  MoveL 7109 to (-196.28, 113.55, -59.38) mm, rotated rx -180 ry 0 rz 0.01 deg; joints [33.121, -44.409, 105.937, -143.593, 67.066, 164.943]
  MoveL 7110 to (-202.77, 114.78, -59.62) mm, rotated rx 180 ry 0 rz 0.01 deg; joints [33.024, -44.143, 105.375, -143.62, 66.8, 164.793]
  MoveL 7111 to (-206.5, 109.33, -59.86) mm, rotated rx 180 ry 0 rz 0.01 deg; joints [32.769, -44.118, 105.358, -143.888, 66.734, 164.906]
  MoveL 7112 to (-202.99, 103.73, -60.11) mm, rotated rx -180 ry 0 rz 0.01 deg; joints [32.66, -44.348, 105.903, -144.081, 66.958, 165.153]
  MoveL 7113 to (-196.46, 104.7, -60.35) mm, rotated rx 180 ry 0 rz 0.01 deg; joints [32.829, -44.542, 106.356, -143.969, 67.215, 165.248]
  MoveL 7114 to (-194.73, 111.07, -60.6) mm, rotated rx 180 ry 0 rz 0.01 deg; joints [33.074, -44.451, 106.172, -143.69, 67.208, 165.087]
  MoveL 7115 to (-199.87, 115.21, -60.84) mm, rotated rx 180 ry 0 rz 0.01 deg; joints [33.1, -44.169, 105.569, -143.583, 66.956, 164.869]
  MoveL 7116 to (-205.73, 112.16, -61.08) mm, rotated rx 180 ry 0 rz 0.01 deg; joints [32.878, -44.018, 105.268, -143.777, 66.773, 164.866]
  MoveL 7117 to (-205.28, 105.57, -61.33) mm, rotated rx -180 ry 0 rz 0.01 deg; joints [32.673, -44.163, 105.628, -144.045, 66.889, 165.09]
  MoveL 7118 to (-199.06, 103.34, -61.57) mm, rotated rx 180 ry 0 rz 0.01 deg; joints [32.731, -44.414, 106.215, -144.068, 67.177, 165.28]
  MoveL 7119 to (-194.53, 108.15, -61.82) mm, rotated rx 180 ry 0 rz 0.01 deg; joints [32.984, -44.455, 106.324, -143.821, 67.302, 165.219]
  MoveL 7120 to (-197.11, 114.22, -62.06) mm, rotated rx 180 ry 0 rz 0.01 deg; joints [33.127, -44.221, 105.822, -143.606, 67.126, 164.988]
  MoveL 7121 to (-203.72, 114.29, -62.3) mm, rotated rx 180 ry 0 rz 0.01 deg; joints [32.99, -43.977, 105.309, -143.681, 66.871, 164.872]
  MoveL 7122 to (-206.42, 108.27, -62.55) mm, rotated rx -180 ry 0 rz 0.01 deg; joints [32.737, -43.999, 105.398, -143.961, 66.853, 165.021]
  MoveL 7123 to (-201.99, 103.37, -62.79) mm, rotated rx -180 ry 0 rz 0.01 deg; joints [32.671, -44.246, 105.98, -144.114, 67.106, 165.263]
  MoveL 7124 to (-195.73, 105.47, -63.04) mm, rotated rx 180 ry 0 rz 0.01 deg; joints [32.871, -44.405, 106.356, -143.958, 67.337, 165.318]
  MoveL 7125 to (-195.14, 112.05, -63.28) mm, rotated rx 180 ry 0 rz 0.01 deg; joints [33.099, -44.27, 106.072, -143.685, 67.28, 165.129]
  MoveL 7126 to (-200.94, 115.22, -63.52) mm, rotated rx 180 ry 0 rz 0.01 deg; joints [33.079, -43.988, 105.468, -143.625, 67.016, 164.93]
  MoveL 7127 to (-206.16, 111.18, -63.77) mm, rotated rx -180 ry 0 rz 0.01 deg; joints [32.838, -43.88, 105.264, -143.852, 66.87, 164.969]
  MoveL 7128 to (-204.56, 104.78, -64.01) mm, rotated rx 180 ry 0 rz 0.01 deg; joints [32.664, -44.06, 105.704, -144.099, 67.031, 165.208]
  MoveL 7129 to (-198.05, 103.68, -64.26) mm, rotated rx 180 ry 0 rz 0.01 deg; joints [32.765, -44.297, 106.258, -144.072, 67.316, 165.368]
  MoveL 7130 to (-194.43, 109.21, -64.5) mm, rotated rx 180 ry 0 rz 0.01 deg; joints [33.022, -44.29, 106.26, -143.807, 67.394, 165.268]
  MoveC 7131 to (-196.76, 111.53, -64.5) mm, rotated rx 180 ry 0 rz 0.01 deg; joints [33.048, -44.16, 105.966, -143.739, 67.27, 165.152] to (-199.08, 109.21, -64.5) mm, rotated rx 180 ry 0 rz 0.01 deg; joints [32.923, -44.129, 105.903, -143.861, 67.209, 165.183]
  MoveC 7132 to (-196.76, 106.88, -64.5) mm, rotated rx 180 ry 0 rz 0.01 deg; joints [32.897, -44.26, 106.197, -143.929, 67.333, 165.299] to (-194.43, 109.21, -64.5) mm, rotated rx -180 ry 0 rz 0.01 deg; joints [33.022, -44.29, 106.26, -143.807, 67.394, 165.268]
  MoveC 7133 to (-193.87, 111.26, -64.5) mm, rotated rx 180 ry 0 rz 0.01 deg; joints [33.1, -44.265, 106.201, -143.716, 67.389, 165.214] to (-192.35, 112.73, -64.5) mm, rotated rx -180 ry 0 rz 0.01 deg; joints [33.181, -44.286, 106.244, -143.638, 67.429, 165.195]
  MoveC 7134 to (-191.13, 114.78, -64.5) mm, rotated rx -180 ry 0 rz 0.01 deg; joints [33.273, -44.283, 106.235, -143.54, 67.449, 165.153] to (-192.33, 116.83, -64.5) mm, rotated rx -180 ry 0 rz 0.01 deg; joints [33.315, -44.198, 106.04, -143.471, 67.374, 165.066]
  MoveC 7135 to (-193.08, 117.28, -64.5) mm, rotated rx -180 ry 0 rz 0.01 deg; joints [33.313, -44.162, 105.96, -143.461, 67.337, 165.038] to (-193.81, 117.76, -64.5) mm, rotated rx -180 ry 0 rz 0.01 deg; joints [33.313, -44.126, 105.88, -143.45, 67.302, 165.009]
  MoveC 7136 to (-196.76, 118.7, -64.5) mm, rotated rx -180 ry 0 rz 0.01 deg; joints [33.281, -44.004, 105.608, -143.446, 67.172, 164.926] to (-199.7, 117.76, -64.5) mm, rotated rx 180 ry 0 rz 0.01 deg; joints [33.188, -43.923, 105.429, -143.518, 67.067, 164.901]
  MoveC 7137 to (-201.1, 116.87, -64.5) mm, rotated rx 180 ry 0 rz 0.01 deg; joints [33.13, -43.893, 105.365, -143.57, 67.023, 164.904] to (-202.59, 116.12, -64.5) mm, rotated rx 180 ry 0 rz 0.01 deg; joints [33.074, -43.858, 105.289, -143.618, 66.974, 164.9]
  MoveC 7138 to (-204.95, 114.01, -64.5) mm, rotated rx -180 ry 0 rz 0.01 deg; joints [32.956, -43.821, 105.212, -143.731, 66.908, 164.924] to (-205.64, 110.92, -64.5) mm, rotated rx 180 ry 0 rz 0.01 deg; joints [32.841, -43.864, 105.313, -143.865, 66.923, 165.009]
  MoveC 7139 to (-205.56, 109.27, -64.5) mm, rotated rx -180 ry 0 rz 0.01 deg; joints [32.789, -43.903, 105.401, -143.932, 66.948, 165.063] to (-205.65, 107.61, -64.5) mm, rotated rx -180 ry 0 rz 0.01 deg; joints [32.733, -43.935, 105.476, -144.001, 66.967, 165.113]
  MoveC 7140 to (-205, 104.51, -64.5) mm, rotated rx 180 ry 0 rz 0.01 deg; joints [32.646, -44.024, 105.68, -144.12, 67.036, 165.223] to (-202.66, 102.37, -64.5) mm, rotated rx -180 ry 0 rz 0.01 deg; joints [32.625, -44.151, 105.966, -144.182, 67.158, 165.333]
  MoveC 7141 to (-201.23, 101.62, -64.5) mm, rotated rx -180 ry 0 rz 0.01 deg; joints [32.63, -44.217, 106.113, -144.196, 67.226, 165.382] to (-199.87, 100.74, -64.5) mm, rotated rx 180 ry 0 rz 0.01 deg; joints [32.63, -44.283, 106.261, -144.217, 67.293, 165.434]
  MoveC 7142 to (-196.86, 99.74, -64.5) mm, rotated rx 180 ry 0 rz 0.01 deg; joints [32.66, -44.408, 106.541, -144.223, 67.427, 165.52] to (-193.81, 100.62, -64.5) mm, rotated rx -180 ry 0 rz 0.01 deg; joints [32.754, -44.494, 106.731, -144.151, 67.536, 165.547]
  MoveC 7143 to (-193.08, 101.1, -64.5) mm, rotated rx -180 ry 0 rz 0.01 deg; joints [32.785, -44.509, 106.763, -144.122, 67.559, 165.546] to (-192.33, 101.56, -64.5) mm, rotated rx 180 ry 0 rz 0.01 deg; joints [32.816, -44.525, 106.798, -144.095, 67.582, 165.545]
  MoveC 7144 to (-191.57, 102, -64.5) mm, rotated rx 180 ry 0 rz 0.01 deg; joints [32.846, -44.542, 106.834, -144.068, 67.607, 165.545] to (-190.79, 102.39, -64.5) mm, rotated rx 180 ry 0 rz 0.01 deg; joints [32.876, -44.561, 106.875, -144.042, 67.632, 165.547]
  MoveC 7145 to (-188.5, 104.54, -64.5) mm, rotated rx -180 ry 0 rz 0.01 deg; joints [32.995, -44.594, 106.944, -143.927, 67.694, 165.521] to (-187.86, 107.61, -64.5) mm, rotated rx -180 ry 0 rz 0.01 deg; joints [33.109, -44.55, 106.841, -143.794, 67.677, 165.437]
  MoveC 7146 to (-187.95, 109.27, -64.5) mm, rotated rx -180 ry 0 rz 0.01 deg; joints [33.162, -44.511, 106.752, -143.727, 67.651, 165.384] to (-187.87, 110.92, -64.5) mm, rotated rx -180 ry 0 rz 0.01 deg; joints [33.217, -44.478, 106.675, -143.659, 67.631, 165.333]
  MoveC 7147 to (-188.56, 114.01, -64.5) mm, rotated rx 180 ry 0 rz 0.01 deg; joints [33.304, -44.388, 106.469, -143.541, 67.562, 165.224] to (-190.92, 116.12, -64.5) mm, rotated rx 180 ry 0 rz 0.01 deg; joints [33.322, -44.261, 106.183, -143.483, 67.439, 165.114]
  MoveC 7148 to (-191.64, 116.46, -64.5) mm, rotated rx -180 ry 0 rz 0.01 deg; joints [33.318, -44.23, 106.112, -143.477, 67.406, 165.09] to (-192.33, 116.83, -64.5) mm, rotated rx 180 ry 0 rz 0.01 deg; joints [33.315, -44.198, 106.04, -143.471, 67.374, 165.066]
  MoveL 7149 to (-192.94, 116.99, -64.33) mm, rotated rx -180 ry 0 rz 0.01 deg; joints [33.307, -44.183, 105.987, -143.469, 67.341, 165.045]
  MoveL 7150 to (-193.39, 116.91, -63.87) mm, rotated rx 180 ry 0 rz 0.01 deg; joints [33.294, -44.194, 105.96, -143.473, 67.306, 165.025]
  MoveL 7151 to (-193.55, 116.84, -63.23) mm, rotated rx -180 ry 0 rz 0.01 deg; joints [33.288, -44.224, 105.956, -143.47, 67.277, 165.005]
  Set speed (1000.0 mm/s)
  MoveL 7152 to (-193.55, 116.84, 11) mm, rotated rx 180 ry 0 rz 0.01 deg; joints [33.247, -48.144, 106.249, -142.533, 64.368, 162.631]
  Set speed (1000.0 mm/s)
  MoveL 7153 to (-195.99, 9.51, 11) mm, rotated rx 180 ry 0 rz 0.01 deg; joints [29.569, -50.402, 111.087, -147.115, 65.397, 165.962]
  Set speed (1000.0 mm/s)
  MoveL 7154 to (-195.99, 9.51, -42.73) mm, rotated rx -180 ry 0 rz 0.01 deg; joints [29.603, -47.446, 110.916, -147.729, 67.753, 167.582]
  Set speed (100.0 mm/s)
  MoveL 7155 to (-196.15, 9.53, -43.35) mm, rotated rx 180 ry 0 rz 0.01 deg; joints [29.601, -47.405, 110.899, -147.736, 67.773, 167.597]
  MoveL 7156 to (-196.59, 9.56, -43.82) mm, rotated rx 180 ry 0 rz 0.01 deg; joints [29.593, -47.363, 110.861, -147.745, 67.774, 167.603]
  MoveL 7157 to (-197.21, 9.55, -44) mm, rotated rx 180 ry 0 rz 0.01 deg; joints [29.58, -47.331, 110.814, -147.755, 67.758, 167.598]
  MoveL 7158 to (-202.45, 5.52, -44.24) mm, rotated rx 180 ry 0 rz 0.01 deg; joints [29.336, -47.21, 110.584, -147.988, 67.608, 167.636]
  MoveL 7159 to (-200.86, -0.89, -44.49) mm, rotated rx 180 ry 0 rz 0.01 deg; joints [29.142, -47.371, 110.981, -148.243, 67.762, 167.85]
  MoveL 7160 to (-194.35, -2, -44.73) mm, rotated rx 180 ry 0 rz 0.01 deg; joints [29.231, -47.605, 111.527, -148.216, 68.049, 167.992]
  MoveL 7161 to (-190.72, 3.52, -44.98) mm, rotated rx -180 ry 0 rz 0.01 deg; joints [29.498, -47.615, 111.567, -147.942, 68.136, 167.901]
  MoveL 7162 to (-194.32, 9.05, -45.22) mm, rotated rx 180 ry 0 rz 0.01 deg; joints [29.621, -47.373, 111.05, -147.754, 67.932, 167.694]
  MoveL 7163 to (-200.84, 7.97, -45.46) mm, rotated rx 180 ry 0 rz 0.01 deg; joints [29.454, -47.152, 110.595, -147.879, 67.694, 167.627]
  MoveL 7164 to (-202.46, 1.57, -45.71) mm, rotated rx 180 ry 0 rz 0.01 deg; joints [29.198, -47.201, 110.746, -148.17, 67.72, 167.79]
  MoveL 7165 to (-197.24, -2.48, -45.95) mm, rotated rx -180 ry 0 rz 0.01 deg; joints [29.158, -47.444, 111.319, -148.283, 67.991, 167.994]
  MoveL 7166 to (-191.44, 0.67, -46.2) mm, rotated rx 180 ry 0 rz 0.01 deg; joints [29.384, -47.574, 111.627, -148.083, 68.195, 168.005]
  MoveL 7167 to (-192.01, 7.25, -46.44) mm, rotated rx -180 ry 0 rz 0.01 deg; joints [29.605, -47.418, 111.298, -147.815, 68.1, 167.817]
  MoveL 7168 to (-198.26, 9.37, -46.68) mm, rotated rx -180 ry 0 rz 0.01 deg; joints [29.555, -47.147, 110.725, -147.802, 67.833, 167.664]
  MoveL 7169 to (-202.71, 4.49, -46.93) mm, rotated rx 180 ry 0 rz 0.01 deg; joints [29.296, -47.07, 110.593, -148.062, 67.725, 167.738]
  MoveL 7170 to (-200.02, -1.54, -47.17) mm, rotated rx 180 ry 0 rz 0.01 deg; joints [29.137, -47.262, 111.059, -148.288, 67.92, 167.958]
  MoveL 7171 to (-193.41, -1.49, -47.42) mm, rotated rx -180 ry 0 rz 0.01 deg; joints [29.269, -47.477, 111.562, -148.21, 68.196, 168.069]
  MoveL 7172 to (-190.81, 4.58, -47.66) mm, rotated rx 180 ry 0 rz 0.01 deg; joints [29.536, -47.441, 111.498, -147.926, 68.234, 167.947]
  MoveL 7173 to (-195.33, 9.39, -47.9) mm, rotated rx -180 ry 0 rz 0.01 deg; joints [29.615, -47.181, 110.942, -147.779, 68.002, 167.745]
  MoveL 7174 to (-201.55, 7.18, -48.15) mm, rotated rx 180 ry 0 rz 0.01 deg; joints [29.414, -46.992, 110.559, -147.948, 67.79, 167.715]
  MoveL 7175 to (-202.02, 0.59, -48.39) mm, rotated rx -180 ry 0 rz 0.01 deg; joints [29.174, -47.084, 110.805, -148.233, 67.865, 167.901]
  MoveL 7176 to (-196.17, -2.47, -48.64) mm, rotated rx -180 ry 0 rz 0.01 deg; joints [29.181, -47.33, 111.385, -148.297, 68.15, 168.087]
  MoveL 7177 to (-191.02, 1.65, -48.88) mm, rotated rx 180 ry 0 rz 0.01 deg; joints [29.429, -47.418, 111.601, -148.064, 68.316, 168.061]
  MoveL 7178 to (-192.74, 8.03, -49.12) mm, rotated rx -180 ry 0 rz 0.01 deg; joints [29.62, -47.227, 111.193, -147.818, 68.176, 167.861]
  MoveL 7179 to (-199.27, 9.01, -49.37) mm, rotated rx 180 ry 0 rz 0.01 deg; joints [29.524, -46.969, 110.648, -147.857, 67.911, 167.735]
  MoveL 7180 to (-202.78, 3.42, -49.61) mm, rotated rx -180 ry 0 rz 0.01 deg; joints [29.259, -46.937, 110.618, -148.135, 67.85, 167.843]
  MoveL 7181 to (-199.07, -2.04, -49.86) mm, rotated rx 180 ry 0 rz 0.01 deg; joints [29.14, -47.153, 111.137, -148.325, 68.08, 168.063]
  MoveL 7182 to (-192.58, -0.83, -50.1) mm, rotated rx 180 ry 0 rz 0.01 deg; joints [29.311, -47.341, 111.581, -148.199, 68.337, 168.14]
  MoveL 7183 to (-191.09, 5.61, -50.35) mm, rotated rx -180 ry 0 rz 0.01 deg; joints [29.568, -47.26, 111.417, -147.913, 68.326, 167.99]
  MoveL 7184 to (-196.39, 9.55, -50.59) mm, rotated rx -180 ry 0 rz 0.01 deg; joints [29.601, -46.99, 110.839, -147.813, 68.072, 167.801]
  MoveL 7185 to (-202.12, 6.28, -50.83) mm, rotated rx 180 ry 0 rz 0.01 deg; joints [29.373, -46.838, 110.538, -148.02, 67.893, 167.808]
  MoveL 7186 to (-201.42, -0.29, -51.08) mm, rotated rx 180 ry 0 rz 0.01 deg; joints [29.156, -46.97, 110.873, -148.291, 68.015, 168.011]
  MoveL 7187 to (-195.12, -2.28, -51.32) mm, rotated rx 180 ry 0 rz 0.01 deg; joints [29.21, -47.211, 111.441, -148.303, 68.306, 168.175]
  MoveL 7188 to (-190.78, 2.69, -51.57) mm, rotated rx 180 ry 0 rz 0.01 deg; joints [29.472, -47.255, 111.559, -148.044, 68.428, 168.112]
  MoveL 7189 to (-193.59, 8.67, -51.81) mm, rotated rx 180 ry 0 rz 0.01 deg; joints [29.627, -47.034, 111.084, -147.829, 68.248, 167.906]
  MoveL 7190 to (-200.19, 8.48, -52.05) mm, rotated rx -180 ry 0 rz 0.01 deg; joints [29.489, -46.796, 110.584, -147.917, 67.995, 167.811]
  MoveL 7191 to (-202.67, 2.36, -52.3) mm, rotated rx -180 ry 0 rz 0.01 deg; joints [29.226, -46.809, 110.656, -148.206, 67.983, 167.951]
  MoveL 7192 to (-198.05, -2.36, -52.54) mm, rotated rx 180 ry 0 rz 0.01 deg; joints [29.15, -47.042, 111.212, -148.353, 68.241, 168.164]
  MoveL 7193 to (-191.88, -0.02, -52.79) mm, rotated rx 180 ry 0 rz 0.01 deg; joints [29.355, -47.198, 111.584, -148.183, 68.471, 168.205]
  MoveL 7194 to (-191.54, 6.57, -53.03) mm, rotated rx 180 ry 0 rz 0.01 deg; joints [29.595, -47.075, 111.324, -147.904, 68.41, 168.033]
  MoveL 7195 to (-197.45, 9.52, -53.27) mm, rotated rx 180 ry 0 rz 0.01 deg; joints [29.58, -46.803, 110.742, -147.853, 68.144, 167.861]
  MoveL 7196 to (-202.52, 5.29, -53.52) mm, rotated rx 180 ry 0 rz 0.01 deg; joints [29.332, -46.692, 110.533, -148.093, 68.003, 167.905]
  MoveL 7197 to (-200.68, -1.05, -53.76) mm, rotated rx 180 ry 0 rz 0.01 deg; joints [29.146, -46.859, 110.947, -148.341, 68.17, 168.12]
  MoveL 7198 to (-194.13, -1.9, -54.01) mm, rotated rx 180 ry 0 rz 0.01 deg; joints [29.245, -47.086, 111.485, -148.301, 68.457, 168.256]
  MoveL 7199 to (-190.72, 3.76, -54.25) mm, rotated rx -180 ry 0 rz 0.01 deg; joints [29.513, -47.085, 111.5, -148.025, 68.532, 168.159]
  MoveL 7200 to (-194.55, 9.14, -54.49) mm, rotated rx -180 ry 0 rz 0.01 deg; joints [29.626, -46.841, 110.973, -147.847, 68.318, 167.953]
  MoveL 7201 to (-201.01, 7.8, -54.74) mm, rotated rx 180 ry 0 rz 0.01 deg; joints [29.45, -46.629, 110.533, -147.982, 68.084, 167.893]
  MoveL 7202 to (-202.37, 1.34, -54.98) mm, rotated rx -180 ry 0 rz 0.01 deg; joints [29.197, -46.688, 110.706, -148.272, 68.123, 168.06]
  MoveL 7203 to (-197, -2.5, -55.23) mm, rotated rx -180 ry 0 rz 0.01 deg; joints [29.168, -46.929, 111.282, -148.373, 68.401, 168.261]
  MoveL 7204 to (-191.33, 0.89, -55.47) mm, rotated rx 180 ry 0 rz 0.01 deg; joints [29.4, -47.048, 111.57, -148.165, 68.597, 168.264]
  MoveL 7205 to (-192.16, 7.44, -55.71) mm, rotated rx -180 ry 0 rz 0.01 deg; joints [29.615, -46.885, 111.222, -147.902, 68.488, 168.075]
  MoveL 7206 to (-198.5, 9.3, -55.96) mm, rotated rx -180 ry 0 rz 0.01 deg; joints [29.554, -46.62, 110.654, -147.902, 68.218, 167.926]
  MoveL 7207 to (-202.74, 4.25, -56.2) mm, rotated rx 180 ry 0 rz 0.01 deg; joints [29.293, -46.553, 110.544, -148.166, 68.122, 168.006]
  MoveL 7208 to (-199.81, -1.67, -56.45) mm, rotated rx 180 ry 0 rz 0.01 deg; joints [29.142, -46.748, 111.023, -148.383, 68.328, 168.226]
  MoveL 7209 to (-193.21, -1.35, -56.69) mm, rotated rx 180 ry 0 rz 0.01 deg; joints [29.284, -46.955, 111.514, -148.294, 68.602, 168.331]
  MoveL 7210 to (-190.86, 4.82, -56.93) mm, rotated rx -180 ry 0 rz 0.01 deg; joints [29.549, -46.909, 111.427, -148.008, 68.627, 168.204]
  MoveL 7211 to (-195.57, 9.45, -57.18) mm, rotated rx 180 ry 0 rz 0.01 deg; joints [29.618, -46.649, 110.864, -147.873, 68.387, 168.004]
  MoveL 7212 to (-201.7, 6.98, -57.42) mm, rotated rx 180 ry 0 rz 0.01 deg; joints [29.41, -46.47, 110.498, -148.051, 68.181, 167.98]
  MoveL 7213 to (-201.9, 0.38, -57.67) mm, rotated rx -180 ry 0 rz 0.01 deg; joints [29.175, -46.57, 110.766, -148.333, 68.268, 168.169]
  MoveL 7214 to (-195.93, -2.45, -57.91) mm, rotated rx 180 ry 0 rz 0.01 deg; joints [29.192, -46.813, 111.344, -148.384, 68.558, 168.352]
  MoveL 7215 to (-190.95, 1.89, -58.15) mm, rotated rx 180 ry 0 rz 0.01 deg; joints [29.445, -46.89, 111.538, -148.144, 68.714, 168.319]
  MoveL 7216 to (-192.92, 8.19, -58.4) mm, rotated rx -180 ry 0 rz 0.01 deg; joints [29.627, -46.694, 111.113, -147.906, 68.562, 168.117]
  MoveL 7217 to (-199.49, 8.91, -58.64) mm, rotated rx 180 ry 0 rz 0.01 deg; joints [29.522, -46.442, 110.577, -147.956, 68.297, 167.997]
  MoveL 7218 to (-202.77, 3.18, -58.89) mm, rotated rx -180 ry 0 rz 0.01 deg; joints [29.256, -46.42, 110.57, -148.238, 68.248, 168.111]
  MoveL 7219 to (-198.84, -2.13, -59.13) mm, rotated rx -180 ry 0 rz 0.01 deg; joints [29.147, -46.638, 111.099, -148.417, 68.488, 168.33]
  MoveL 7220 to (-192.41, -0.65, -59.37) mm, rotated rx 180 ry 0 rz 0.01 deg; joints [29.327, -46.817, 111.528, -148.28, 68.741, 168.4]
  MoveL 7221 to (-191.18, 5.84, -59.62) mm, rotated rx -180 ry 0 rz 0.01 deg; joints [29.58, -46.727, 111.341, -147.995, 68.716, 168.246]
  MoveL 7222 to (-196.63, 9.56, -59.86) mm, rotated rx 180 ry 0 rz 0.01 deg; joints [29.602, -46.459, 110.76, -147.907, 68.456, 168.059]
  MoveL 7223 to (-202.23, 6.06, -60.11) mm, rotated rx 180 ry 0 rz 0.01 deg; joints [29.369, -46.317, 110.48, -148.122, 68.284, 168.073]
  MoveL 7224 to (-201.26, -0.47, -60.35) mm, rotated rx 180 ry 0 rz 0.01 deg; joints [29.159, -46.456, 110.834, -148.388, 68.42, 168.278]
  MoveL 7225 to (-194.89, -2.21, -60.6) mm, rotated rx 180 ry 0 rz 0.01 deg; joints [29.223, -46.691, 111.396, -148.387, 68.712, 168.437]
  MoveL 7226 to (-190.75, 2.94, -60.84) mm, rotated rx 180 ry 0 rz 0.01 deg; joints [29.487, -46.725, 111.49, -148.124, 68.823, 168.368]
  MoveL 7227 to (-193.8, 8.79, -61.08) mm, rotated rx 180 ry 0 rz 0.01 deg; joints [29.632, -46.5, 111.002, -147.917, 68.632, 168.162]
  MoveL 7228 to (-200.39, 8.34, -61.33) mm, rotated rx 180 ry 0 rz 0.01 deg; joints [29.486, -46.27, 110.514, -148.017, 68.381, 168.073]
  MoveL 7229 to (-202.62, 2.12, -61.57) mm, rotated rx 180 ry 0 rz 0.01 deg; joints [29.224, -46.293, 110.609, -148.306, 68.382, 168.218]
  MoveL 7230 to (-197.81, -2.41, -61.82) mm, rotated rx -180 ry 0 rz 0.01 deg; joints [29.159, -46.526, 111.171, -148.442, 68.648, 168.429]
  MoveL 7231 to (-191.74, 0.18, -62.06) mm, rotated rx -180 ry 0 rz 0.01 deg; joints [29.371, -46.672, 111.525, -148.263, 68.872, 168.463]
  MoveL 7232 to (-191.67, 6.78, -62.3) mm, rotated rx 180 ry 0 rz 0.01 deg; joints [29.605, -46.54, 111.243, -147.988, 68.797, 168.287]
  MoveL 7233 to (-197.69, 9.49, -62.55) mm, rotated rx -180 ry 0 rz 0.01 deg; joints [29.58, -46.272, 110.663, -147.949, 68.527, 168.119]
  MoveL 7234 to (-202.59, 5.05, -62.79) mm, rotated rx 180 ry 0 rz 0.01 deg; joints [29.328, -46.172, 110.477, -148.195, 68.396, 168.17]
  MoveL 7235 to (-200.49, -1.21, -63.04) mm, rotated rx -180 ry 0 rz 0.01 deg; joints [29.15, -46.343, 110.906, -148.435, 68.575, 168.386]
  MoveL 7236 to (-193.91, -1.79, -63.28) mm, rotated rx 180 ry 0 rz 0.01 deg; joints [29.259, -46.564, 111.434, -148.383, 68.861, 168.516]
  MoveL 7237 to (-190.74, 4, -63.52) mm, rotated rx 180 ry 0 rz 0.01 deg; joints [29.527, -46.553, 111.426, -148.104, 68.924, 168.414]
  MoveL 7238 to (-194.77, 9.23, -63.77) mm, rotated rx -180 ry 0 rz 0.01 deg; joints [29.63, -46.307, 110.889, -147.937, 68.701, 168.209]
  MoveL 7239 to (-201.18, 7.63, -64.01) mm, rotated rx 180 ry 0 rz 0.01 deg; joints [29.447, -46.104, 110.465, -148.082, 68.471, 168.155]
  MoveL 7240 to (-202.28, 1.11, -64.26) mm, rotated rx -180 ry 0 rz 0.01 deg; joints [29.197, -46.171, 110.66, -148.37, 68.523, 168.326]
  MoveL 7241 to (-196.75, -2.5, -64.5) mm, rotated rx -180 ry 0 rz 0.01 deg; joints [29.178, -46.411, 111.238, -148.459, 68.807, 168.523]
  MoveL 7242 to (-193.37, -2.5, -64.5) mm, rotated rx 180 ry 0 rz 0.01 deg; joints [29.245, -46.525, 111.497, -148.418, 68.945, 168.578]
  MoveC 7243 to (-192.01, -1.4, -64.5) mm, rotated rx -180 ry 0 rz 0.01 deg; joints [29.311, -46.552, 111.554, -148.356, 68.986, 168.57] to (-192.8, 0.16, -64.5) mm, rotated rx -180 ry 0 rz 0.01 deg; joints [29.351, -46.497, 111.427, -148.3, 68.933, 168.514]
  MoveC 7244 to (-193.54, 0.5, -64.5) mm, rotated rx -180 ry 0 rz 0.01 deg; joints [29.348, -46.466, 111.356, -148.295, 68.898, 168.493] to (-194.28, 0.85, -64.5) mm, rotated rx 180 ry 0 rz 0.01 deg; joints [29.346, -46.434, 111.284, -148.289, 68.863, 168.471]
  MoveC 7245 to (-195.01, 1.21, -64.5) mm, rotated rx 180 ry 0 rz 0.01 deg; joints [29.344, -46.403, 111.213, -148.282, 68.829, 168.449] to (-195.73, 1.6, -64.5) mm, rotated rx -180 ry 0 rz 0.01 deg; joints [29.343, -46.372, 111.141, -148.275, 68.794, 168.426]
  MoveC 7246 to (-196.76, 1.86, -64.5) mm, rotated rx -180 ry 0 rz 0.01 deg; joints [29.332, -46.332, 111.05, -148.276, 68.749, 168.402] to (-197.79, 1.59, -64.5) mm, rotated rx -180 ry 0 rz 0.01 deg; joints [29.302, -46.302, 110.983, -148.3, 68.71, 168.393]
  MoveC 7247 to (-198.49, 1.21, -64.5) mm, rotated rx -180 ry 0 rz 0.01 deg; joints [29.275, -46.285, 110.945, -148.324, 68.687, 168.392] to (-199.21, 0.84, -64.5) mm, rotated rx 180 ry 0 rz 0.01 deg; joints [29.248, -46.267, 110.906, -148.348, 68.662, 168.39]
  MoveC 7248 to (-199.93, 0.49, -64.5) mm, rotated rx 180 ry 0 rz 0.01 deg; joints [29.222, -46.249, 110.866, -148.371, 68.638, 168.388] to (-200.65, 0.16, -64.5) mm, rotated rx 180 ry 0 rz 0.01 deg; joints [29.195, -46.23, 110.824, -148.394, 68.612, 168.386]
  MoveC 7249 to (-201.44, -1.4, -64.5) mm, rotated rx 180 ry 0 rz 0.01 deg; joints [29.125, -46.231, 110.831, -148.468, 68.601, 168.416] to (-200.08, -2.5, -64.5) mm, rotated rx -180 ry 0 rz 0.01 deg; joints [29.113, -46.297, 110.982, -148.498, 68.671, 168.469]
  MoveL 7250 to (-196.75, -2.5, -64.5) mm, rotated rx -180 ry 0 rz 0.01 deg; joints [29.178, -46.411, 111.238, -148.459, 68.807, 168.523]
  MoveC 7251 to (-194.7, -3.12, -64.5) mm, rotated rx -180 ry 0 rz 0.01 deg; joints [29.197, -46.491, 111.422, -148.46, 68.899, 168.574] to (-193.34, -4.77, -64.5) mm, rotated rx -180 ry 0 rz 0.01 deg; joints [29.165, -46.567, 111.596, -148.513, 68.976, 168.641]
  MoveC 7252 to (-191.98, -6.43, -64.5) mm, rotated rx 180 ry 0 rz 0.01 deg; joints [29.134, -46.642, 111.771, -148.566, 69.054, 168.709] to (-189.93, -7.05, -64.5) mm, rotated rx -180 ry 0 rz 0.01 deg; joints [29.152, -46.723, 111.953, -148.567, 69.145, 168.759]
  MoveL 7253 to (-172.26, -7.05, -64.5) mm, rotated rx 180 ry 0 rz 0.01 deg; joints [29.506, -47.313, 113.294, -148.345, 69.861, 169.045]
  MoveC 7254 to (-170.9, -5.95, -64.5) mm, rotated rx 180 ry 0 rz 0.01 deg; joints [29.573, -47.339, 113.35, -148.281, 69.901, 169.037] to (-171.69, -4.39, -64.5) mm, rotated rx 180 ry 0 rz 0.01 deg; joints [29.613, -47.285, 113.224, -148.226, 69.848, 168.982]
  MoveC 7255 to (-177.36, -1.9, -64.5) mm, rotated rx 180 ry 0 rz 0.01 deg; joints [29.587, -47.052, 112.69, -148.194, 69.586, 168.823] to (-183.07, 0.47, -64.5) mm, rotated rx -180 ry 0 rz 0.01 deg; joints [29.556, -46.819, 112.155, -148.167, 69.324, 168.664]
  MoveC 7256 to (-188.72, 3, -64.5) mm, rotated rx -180 ry 0 rz 0.01 deg; joints [29.532, -46.583, 111.616, -148.131, 69.061, 168.502] to (-194.17, 5.94, -64.5) mm, rotated rx 180 ry 0 rz 0.01 deg; joints [29.527, -46.346, 111.073, -148.074, 68.8, 168.331]
  MoveC 7257 to (-196.78, 6.65, -64.5) mm, rotated rx 180 ry 0 rz 0.01 deg; joints [29.5, -46.244, 110.842, -148.076, 68.684, 168.268] to (-199.38, 5.92, -64.5) mm, rotated rx 180 ry 0 rz 0.01 deg; joints [29.423, -46.169, 110.674, -148.137, 68.588, 168.246]
  MoveC 7258 to (-204.79, 2.96, -64.5) mm, rotated rx 180 ry 0 rz 0.01 deg; joints [29.213, -46.038, 110.385, -148.325, 68.406, 168.24] to (-210.43, 0.44, -64.5) mm, rotated rx 180 ry 0 rz 0.01 deg; joints [29.014, -45.89, 110.057, -148.495, 68.207, 168.217]
  MoveC 7259 to (-216.13, -1.91, -64.5) mm, rotated rx 180 ry 0 rz 0.01 deg; joints [28.821, -45.735, 109.715, -148.658, 68.003, 168.189] to (-221.77, -4.39, -64.5) mm, rotated rx 180 ry 0 rz 0.01 deg; joints [28.627, -45.584, 109.38, -148.824, 67.802, 168.166]
  MoveC 7260 to (-222.56, -5.95, -64.5) mm, rotated rx 180 ry 0 rz 0.01 deg; joints [28.557, -45.584, 109.384, -148.898, 67.79, 168.196] to (-221.2, -7.05, -64.5) mm, rotated rx -180 ry 0 rz 0.01 deg; joints [28.544, -45.651, 109.538, -148.93, 67.86, 168.249]
  MoveL 7261 to (-189.93, -7.05, -64.5) mm, rotated rx -180 ry 0 rz 0.01 deg; joints [29.152, -46.723, 111.953, -148.567, 69.145, 168.759]
  MoveC 7262 to (-187.1, -7.91, -64.5) mm, rotated rx -180 ry 0 rz 0.01 deg; joints [29.178, -46.833, 112.206, -148.569, 69.272, 168.829] to (-185.22, -10.19, -64.5) mm, rotated rx 180 ry 0 rz 0.01 deg; joints [29.134, -46.937, 112.446, -148.641, 69.379, 168.921]
  MoveC 7263 to (-183.34, -12.48, -64.5) mm, rotated rx -180 ry 0 rz 0.01 deg; joints [29.09, -47.04, 112.686, -148.714, 69.486, 169.014] to (-180.5, -13.33, -64.5) mm, rotated rx 180 ry 0 rz 0.01 deg; joints [29.115, -47.15, 112.937, -148.715, 69.613, 169.082]
  MoveL 7264 to (-143.07, -13.33, -64.5) mm, rotated rx -180 ry 0 rz 0.01 deg; joints [29.881, -48.376, 115.74, -148.214, 71.115, 169.683]
  MoveC 7265 to (-141.71, -12.24, -64.5) mm, rotated rx 180 ry 0 rz 0.01 deg; joints [29.949, -48.401, 115.794, -148.149, 71.154, 169.675] to (-142.49, -10.67, -64.5) mm, rotated rx 180 ry 0 rz 0.01 deg; joints [29.989, -48.348, 115.669, -148.094, 71.101, 169.621]
  MoveL 7266 to (-188.98, 10.13, -64.5) mm, rotated rx -180 ry 0 rz 0.01 deg; joints [29.778, -46.445, 111.288, -147.836, 68.955, 168.3]
  MoveC 7267 to (-190.22, 10.77, -64.5) mm, rotated rx -180 ry 0 rz 0.01 deg; joints [29.776, -46.391, 111.165, -147.824, 68.896, 168.261] to (-191.4, 11.54, -64.5) mm, rotated rx 180 ry 0 rz 0.01 deg; joints [29.779, -46.338, 111.042, -147.806, 68.838, 168.221]
  MoveC 7268 to (-192.52, 12.36, -64.5) mm, rotated rx -180 ry 0 rz 0.01 deg; joints [29.785, -46.284, 110.92, -147.785, 68.781, 168.179] to (-193.65, 13.19, -64.5) mm, rotated rx 180 ry 0 rz 0.01 deg; joints [29.792, -46.231, 110.798, -147.764, 68.724, 168.137]
  MoveC 7269 to (-196.67, 14.21, -64.5) mm, rotated rx 180 ry 0 rz 0.01 deg; joints [29.767, -46.109, 110.521, -147.758, 68.588, 168.058] to (-199.72, 13.27, -64.5) mm, rotated rx 180 ry 0 rz 0.01 deg; joints [29.673, -46.023, 110.328, -147.834, 68.476, 168.034]
  MoveC 7270 to (-200.95, 12.4, -64.5) mm, rotated rx -180 ry 0 rz 0.01 deg; joints [29.619, -45.997, 110.272, -147.885, 68.438, 168.038] to (-202.16, 11.51, -64.5) mm, rotated rx 180 ry 0 rz 0.01 deg; joints [29.564, -45.972, 110.218, -147.936, 68.4, 168.043]
  MoveC 7271 to (-203.41, 10.68, -64.5) mm, rotated rx -180 ry 0 rz 0.01 deg; joints [29.51, -45.944, 110.157, -147.985, 68.36, 168.046] to (-204.75, 9.99, -64.5) mm, rotated rx -180 ry 0 rz 0.01 deg; joints [29.459, -45.911, 110.084, -148.03, 68.314, 168.043]
  MoveL 7272 to (-250.99, -10.68, -64.5) mm, rotated rx 180 ry 0 rz 0.01 deg; joints [27.861, -44.664, 107.335, -149.39, 66.659, 167.86]
  MoveC 7273 to (-251.78, -12.24, -64.5) mm, rotated rx 180 ry 0 rz 0.01 deg; joints [27.792, -44.663, 107.337, -149.463, 66.646, 167.891] to (-250.42, -13.33, -64.5) mm, rotated rx 180 ry 0 rz 0.01 deg; joints [27.779, -44.732, 107.492, -149.496, 66.717, 167.945]
  MoveL 7274 to (-180.5, -13.33, -64.5) mm, rotated rx 180 ry 0 rz 0.01 deg; joints [29.115, -47.15, 112.937, -148.715, 69.613, 169.082]
  MoveC 7275 to (-177.67, -14.19, -64.5) mm, rotated rx 180 ry 0 rz 0.01 deg; joints [29.141, -47.26, 113.188, -148.715, 69.739, 169.151] to (-175.79, -16.48, -64.5) mm, rotated rx 180 ry 0 rz 0.01 deg; joints [29.097, -47.362, 113.427, -148.787, 69.846, 169.243]
  MoveC 7276 to (-173.91, -18.76, -64.5) mm, rotated rx 180 ry 0 rz 0.01 deg; joints [29.052, -47.464, 113.665, -148.859, 69.953, 169.334] to (-171.07, -19.62, -64.5) mm, rotated rx -180 ry 0 rz 0.01 deg; joints [29.078, -47.573, 113.914, -148.859, 70.079, 169.402]
  MoveL 7277 to (-113.87, -19.62, -64.5) mm, rotated rx -180 ry 0 rz 0.01 deg; joints [30.271, -49.408, 118.141, -148.05, 72.355, 170.313]
  MoveC 7278 to (-112.51, -18.52, -64.5) mm, rotated rx -180 ry 0 rz 0.01 deg; joints [30.341, -49.432, 118.193, -147.983, 72.393, 170.307] to (-113.3, -16.96, -64.5) mm, rotated rx 180 ry 0 rz 0.01 deg; joints [30.382, -49.381, 118.07, -147.929, 72.34, 170.254]
  MoveL 7279 to (-186.46, 15.7, -64.5) mm, rotated rx 180 ry 0 rz 0.01 deg; joints [30.024, -46.427, 111.236, -147.572, 68.982, 168.185]
  MoveC 7280 to (-188.9, 17.07, -64.5) mm, rotated rx -180 ry 0 rz 0.01 deg; joints [30.023, -46.32, 110.99, -147.545, 68.865, 168.107] to (-191.06, 18.84, -64.5) mm, rotated rx -180 ry 0 rz 0.01 deg; joints [30.041, -46.214, 110.748, -147.497, 68.754, 168.021]
  MoveC 7281 to (-192.98, 20.87, -64.5) mm, rotated rx -180 ry 0 rz 0.01 deg; joints [30.073, -46.111, 110.512, -147.436, 68.649, 167.931] to (-194.74, 23.02, -64.5) mm, rotated rx 180 ry 0 rz 0.01 deg; joints [30.113, -46.011, 110.282, -147.367, 68.549, 167.841]
  MoveC 7282 to (-196.82, 24.04, -64.5) mm, rotated rx 180 ry 0 rz 0.01 deg; joints [30.106, -45.921, 110.077, -147.35, 68.451, 167.777] to (-198.86, 22.95, -64.5) mm, rotated rx 180 ry 0 rz 0.01 deg; joints [30.027, -45.872, 109.969, -147.42, 68.382, 167.774]
  MoveC 7283 to (-199.83, 21.64, -64.5) mm, rotated rx 180 ry 0 rz 0.01 deg; joints [29.962, -45.863, 109.952, -147.486, 68.36, 167.795] to (-200.87, 20.38, -64.5) mm, rotated rx 180 ry 0 rz 0.01 deg; joints [29.898, -45.852, 109.928, -147.551, 68.335, 167.813]
  MoveC 7284 to (-202.01, 19.21, -64.5) mm, rotated rx -180 ry 0 rz 0.01 deg; joints [29.835, -45.834, 109.892, -147.613, 68.304, 167.827] to (-203.29, 18.2, -64.5) mm, rotated rx -180 ry 0 rz 0.01 deg; joints [29.774, -45.809, 109.838, -147.67, 68.265, 167.835]
  MoveC 7285 to (-204.26, 17.51, -64.5) mm, rotated rx 180 ry 0 rz 0.01 deg; joints [29.731, -45.789, 109.793, -147.71, 68.235, 167.838] to (-205.22, 16.79, -64.5) mm, rotated rx 180 ry 0 rz 0.01 deg; joints [29.687, -45.769, 109.751, -147.751, 68.205, 167.843]
  MoveC 7286 to (-206.21, 16.12, -64.5) mm, rotated rx 180 ry 0 rz 0.01 deg; joints [29.644, -45.747, 109.704, -147.79, 68.173, 167.845] to (-207.27, 15.57, -64.5) mm, rotated rx 180 ry 0 rz 0.01 deg; joints [29.604, -45.721, 109.646, -147.826, 68.137, 167.843]
  MoveL 7287 to (-280.21, -16.96, -64.5) mm, rotated rx 180 ry 0 rz 0.01 deg; joints [27.118, -43.713, 105.234, -149.921, 65.491, 167.552]
  MoveC 7288 to (-281, -18.52, -64.5) mm, rotated rx 180 ry 0 rz 0.01 deg; joints [27.051, -43.712, 105.234, -149.994, 65.476, 167.584] to (-279.64, -19.62, -64.5) mm, rotated rx -180 ry 0 rz 0.01 deg; joints [27.037, -43.782, 105.391, -150.028, 65.549, 167.638]
  MoveL 7289 to (-171.07, -19.62, -64.5) mm, rotated rx -180 ry 0 rz 0.01 deg; joints [29.078, -47.573, 113.914, -148.859, 70.079, 169.402]
  MoveL 7290 to (-170.46, -19.47, -64.33) mm, rotated rx -180 ry 0 rz 0.01 deg; joints [29.096, -47.6, 113.955, -148.843, 70.094, 169.403]
  MoveL 7291 to (-170.11, -19.17, -63.87) mm, rotated rx 180 ry 0 rz 0.01 deg; joints [29.113, -47.634, 113.973, -148.822, 70.084, 169.388]
  MoveL 7292 to (-170, -19.04, -63.23) mm, rotated rx 180 ry 0 rz 0.01 deg; joints [29.12, -47.672, 113.98, -148.809, 70.058, 169.368]
  Set speed (1000.0 mm/s)
  MoveL 7293 to (-170, -19.04, 11) mm, rotated rx 180 ry 0 rz 0.01 deg; joints [29.071, -51.925, 114.283, -148.04, 66.682, 167.163]
  Set speed (1000.0 mm/s)
  MoveL 7294 to (-328.23, 254.06, 11) mm, rotated rx -180 ry 0 rz 0.01 deg; joints [34.658, -39.098, 87.572, -137.594, 57.514, 154.821]
  Set speed (1000.0 mm/s)
  MoveL 7295 to (-328.23, 254.06, -42.73) mm, rotated rx -180 ry 0 rz 0.01 deg; joints [34.683, -36.67, 87.401, -138.497, 59.203, 156.58]
  Set speed (100.0 mm/s)
  MoveL 7296 to (-328.07, 254.04, -43.35) mm, rotated rx -180 ry 0 rz 0.01 deg; joints [34.686, -36.649, 87.414, -138.507, 59.23, 156.604]
  MoveL 7297 to (-327.62, 254.01, -43.82) mm, rotated rx -180 ry 0 rz 0.01 deg; joints [34.694, -36.647, 87.453, -138.515, 59.264, 156.631]
  MoveL 7298 to (-327, 254.02, -44) mm, rotated rx -180 ry 0 rz 0.01 deg; joints [34.707, -36.664, 87.506, -138.515, 59.296, 156.652]
  MoveL 7299 to (-321.77, 258.05, -44.24) mm, rotated rx 180 ry 0 rz 0.01 deg; joints [34.924, -36.759, 87.722, -138.334, 59.478, 156.626]
  MoveL 7300 to (-323.36, 264.46, -44.49) mm, rotated rx -180 ry 0 rz 0.01 deg; joints [35.074, -36.496, 87.18, -138.066, 59.333, 156.328]
  MoveL 7301 to (-329.87, 265.57, -44.73) mm, rotated rx 180 ry 0 rz 0.01 deg; joints [34.977, -36.174, 86.525, -138.035, 59.043, 156.122]
  MoveL 7302 to (-333.5, 260.05, -44.98) mm, rotated rx -180 ry 0 rz 0.01 deg; joints [34.751, -36.168, 86.542, -138.284, 58.965, 156.266]
  MoveL 7303 to (-329.89, 254.52, -45.22) mm, rotated rx -180 ry 0 rz 0.01 deg; joints [34.665, -36.471, 87.21, -138.519, 59.202, 156.596]
  MoveL 7304 to (-323.38, 255.6, -45.46) mm, rotated rx 180 ry 0 rz 0.01 deg; joints [34.823, -36.705, 87.724, -138.462, 59.478, 156.724]
  MoveL 7305 to (-321.76, 262, -45.71) mm, rotated rx 180 ry 0 rz 0.01 deg; joints [35.037, -36.578, 87.469, -138.187, 59.471, 156.509]
  MoveL 7306 to (-326.98, 266.05, -45.95) mm, rotated rx 180 ry 0 rz 0.01 deg; joints [35.048, -36.228, 86.748, -138.028, 59.2, 156.215]
  MoveL 7307 to (-332.78, 262.89, -46.2) mm, rotated rx -180 ry 0 rz 0.01 deg; joints [34.845, -36.06, 86.422, -138.179, 58.996, 156.204]
  MoveL 7308 to (-332.21, 256.31, -46.44) mm, rotated rx 180 ry 0 rz 0.01 deg; joints [34.671, -36.264, 86.883, -138.466, 59.114, 156.5]
  MoveL 7309 to (-325.95, 254.2, -46.68) mm, rotated rx 180 ry 0 rz 0.01 deg; joints [34.734, -36.579, 87.574, -138.547, 59.422, 156.755]
  MoveL 7310 to (-321.51, 259.08, -46.93) mm, rotated rx 180 ry 0 rz 0.01 deg; joints [34.96, -36.616, 87.666, -138.33, 59.558, 156.674]
  MoveL 7311 to (-324.2, 265.11, -47.17) mm, rotated rx 180 ry 0 rz 0.01 deg; joints [35.077, -36.317, 87.048, -138.082, 59.369, 156.364]
  MoveL 7312 to (-330.8, 265.06, -47.42) mm, rotated rx -180 ry 0 rz 0.01 deg; joints [34.945, -36.025, 86.457, -138.101, 59.09, 156.203]
  MoveL 7313 to (-333.4, 258.99, -47.66) mm, rotated rx 180 ry 0 rz 0.01 deg; joints [34.724, -36.079, 86.602, -138.371, 59.064, 156.396]
  MoveL 7314 to (-328.88, 254.18, -47.9) mm, rotated rx -180 ry 0 rz 0.01 deg; joints [34.676, -36.399, 87.306, -138.574, 59.332, 156.719]
  MoveL 7315 to (-322.66, 256.39, -48.15) mm, rotated rx 180 ry 0 rz 0.01 deg; joints [34.861, -36.588, 87.724, -138.468, 59.581, 156.793]
  MoveL 7316 to (-322.19, 262.98, -48.39) mm, rotated rx -180 ry 0 rz 0.01 deg; joints [35.057, -36.407, 87.354, -138.188, 59.522, 156.542]
  MoveL 7317 to (-328.04, 266.04, -48.64) mm, rotated rx -180 ry 0 rz 0.01 deg; joints [35.028, -36.058, 86.637, -138.073, 59.235, 156.271]
  MoveL 7318 to (-333.2, 261.91, -48.88) mm, rotated rx -180 ry 0 rz 0.01 deg; joints [34.811, -35.947, 86.43, -138.264, 59.072, 156.317]
  MoveL 7319 to (-331.48, 255.54, -49.13) mm, rotated rx 180 ry 0 rz 0.01 deg; joints [34.664, -36.193, 86.982, -138.539, 59.238, 156.634]
  MoveL 7320 to (-324.95, 254.56, -49.37) mm, rotated rx 180 ry 0 rz 0.01 deg; joints [34.765, -36.487, 87.626, -138.571, 59.543, 156.849]
  MoveL 7321 to (-321.43, 260.15, -49.61) mm, rotated rx 180 ry 0 rz 0.01 deg; joints [34.992, -36.464, 87.591, -138.326, 59.629, 156.716]
  MoveL 7322 to (-325.14, 265.61, -49.86) mm, rotated rx -180 ry 0 rz 0.01 deg; joints [35.073, -36.138, 86.917, -138.104, 59.403, 156.402]
  MoveL 7323 to (-331.64, 264.4, -50.1) mm, rotated rx 180 ry 0 rz 0.01 deg; joints [34.911, -35.885, 86.408, -138.173, 59.144, 156.292]
  MoveL 7324 to (-333.13, 257.96, -50.35) mm, rotated rx 180 ry 0 rz 0.01 deg; joints [34.701, -35.997, 86.675, -138.457, 59.171, 156.529]
  MoveL 7325 to (-327.83, 254.02, -50.59) mm, rotated rx 180 ry 0 rz 0.01 deg; joints [34.694, -36.324, 87.395, -138.619, 59.462, 156.835]
  MoveL 7326 to (-322.09, 257.29, -50.83) mm, rotated rx 180 ry 0 rz 0.01 deg; joints [34.899, -36.461, 87.702, -138.468, 59.675, 156.854]
  MoveL 7327 to (-322.79, 263.86, -51.08) mm, rotated rx 180 ry 0 rz 0.01 deg; joints [35.071, -36.231, 87.229, -138.193, 59.565, 156.573]
  MoveL 7328 to (-329.09, 265.85, -51.32) mm, rotated rx 180 ry 0 rz 0.01 deg; joints [35.003, -35.895, 86.539, -138.125, 59.272, 156.336]
  MoveL 7329 to (-333.44, 260.88, -51.57) mm, rotated rx -180 ry 0 rz 0.01 deg; joints [34.778, -35.843, 86.457, -138.351, 59.156, 156.437]
  MoveL 7330 to (-330.62, 254.9, -51.81) mm, rotated rx 180 ry 0 rz 0.01 deg; joints [34.664, -36.123, 87.082, -138.606, 59.366, 156.765]
  MoveL 7331 to (-324.02, 255.08, -52.05) mm, rotated rx -180 ry 0 rz 0.01 deg; joints [34.799, -36.386, 87.66, -138.586, 59.658, 156.933]
  MoveL 7332 to (-321.54, 261.21, -52.3) mm, rotated rx -180 ry 0 rz 0.01 deg; joints [35.021, -36.304, 87.499, -138.322, 59.692, 156.752]
  MoveL 7333 to (-326.16, 265.93, -52.54) mm, rotated rx 180 ry 0 rz 0.01 deg; joints [35.063, -35.961, 86.789, -138.134, 59.436, 156.446]
  MoveL 7334 to (-332.34, 263.59, -52.79) mm, rotated rx -180 ry 0 rz 0.01 deg; joints [34.876, -35.754, 86.379, -138.251, 59.205, 156.39]
  MoveL 7335 to (-332.67, 257, -53.03) mm, rotated rx 180 ry 0 rz 0.01 deg; joints [34.684, -35.919, 86.76, -138.539, 59.286, 156.663]
  MoveL 7336 to (-326.76, 254.05, -53.27) mm, rotated rx -180 ry 0 rz 0.01 deg; joints [34.717, -36.243, 87.472, -138.656, 59.59, 156.944]
  MoveL 7337 to (-321.69, 258.28, -53.52) mm, rotated rx -180 ry 0 rz 0.01 deg; joints [34.936, -36.324, 87.66, -138.466, 59.762, 156.906]
  MoveL 7338 to (-323.54, 264.62, -53.76) mm, rotated rx -180 ry 0 rz 0.01 deg; joints [35.079, -36.053, 87.098, -138.203, 59.604, 156.605]
  MoveL 7339 to (-330.09, 265.47, -54.01) mm, rotated rx 180 ry 0 rz 0.01 deg; joints [34.974, -35.739, 86.456, -138.184, 59.315, 156.408]
  MoveL 7340 to (-333.49, 259.81, -54.25) mm, rotated rx -180 ry 0 rz 0.01 deg; joints [34.748, -35.747, 86.502, -138.438, 59.249, 156.563]
  MoveL 7341 to (-329.67, 254.42, -54.49) mm, rotated rx -180 ry 0 rz 0.01 deg; joints [34.671, -36.052, 87.18, -138.665, 59.496, 156.891]
  MoveL 7342 to (-323.2, 255.77, -54.74) mm, rotated rx 180 ry 0 rz 0.01 deg; joints [34.836, -36.275, 87.673, -138.596, 59.767, 157.008]
  MoveL 7343 to (-321.84, 262.23, -54.98) mm, rotated rx 180 ry 0 rz 0.01 deg; joints [35.046, -36.136, 87.391, -138.32, 59.747, 156.785]
  MoveL 7344 to (-327.22, 266.07, -55.23) mm, rotated rx -180 ry 0 rz 0.01 deg; joints [35.048, -35.787, 86.669, -138.172, 59.469, 156.495]
  MoveL 7345 to (-332.89, 262.68, -55.47) mm, rotated rx -180 ry 0 rz 0.01 deg; joints [34.841, -35.633, 86.369, -138.332, 59.274, 156.496]
  MoveL 7346 to (-332.05, 256.13, -55.71) mm, rotated rx 180 ry 0 rz 0.01 deg; joints [34.673, -35.846, 86.852, -138.616, 59.405, 156.797]
  MoveL 7347 to (-325.72, 254.26, -55.96) mm, rotated rx 180 ry 0 rz 0.01 deg; joints [34.745, -36.155, 87.534, -138.685, 59.715, 157.043]
  MoveL 7348 to (-321.47, 259.32, -56.2) mm, rotated rx 180 ry 0 rz 0.01 deg; joints [34.972, -36.178, 87.597, -138.461, 59.839, 156.951]
  MoveL 7349 to (-324.41, 265.24, -56.45) mm, rotated rx -180 ry 0 rz 0.01 deg; joints [35.08, -35.873, 86.965, -138.219, 59.639, 156.64]
  MoveL 7350 to (-331, 264.92, -56.69) mm, rotated rx 180 ry 0 rz 0.01 deg; joints [34.942, -35.592, 86.39, -138.251, 59.362, 156.489]
  MoveL 7351 to (-333.36, 258.75, -56.93) mm, rotated rx 180 ry 0 rz 0.01 deg; joints [34.722, -35.658, 86.563, -138.524, 59.35, 156.692]
  MoveL 7352 to (-328.65, 254.12, -57.18) mm, rotated rx 180 ry 0 rz 0.01 deg; joints [34.684, -35.979, 87.273, -138.716, 59.626, 157.012]
  MoveL 7353 to (-322.52, 256.59, -57.42) mm, rotated rx 180 ry 0 rz 0.01 deg; joints [34.874, -36.155, 87.666, -138.599, 59.867, 157.074]
  MoveL 7354 to (-322.32, 263.19, -57.67) mm, rotated rx 180 ry 0 rz 0.01 deg; joints [35.065, -35.964, 87.272, -138.32, 59.794, 156.816]
  MoveL 7355 to (-328.28, 266.02, -57.91) mm, rotated rx 180 ry 0 rz 0.01 deg; joints [35.026, -35.619, 86.558, -138.217, 59.503, 156.552]
  MoveL 7356 to (-333.27, 261.68, -58.15) mm, rotated rx 180 ry 0 rz 0.01 deg; joints [34.807, -35.521, 86.38, -138.417, 59.351, 156.61]
  MoveL 7357 to (-331.29, 255.38, -58.4) mm, rotated rx 180 ry 0 rz 0.01 deg; joints [34.668, -35.774, 86.949, -138.687, 59.53, 156.929]
  MoveL 7358 to (-324.73, 254.66, -58.64) mm, rotated rx -180 ry 0 rz 0.01 deg; joints [34.777, -36.06, 87.58, -138.706, 59.834, 157.134]
  MoveL 7359 to (-321.44, 260.39, -58.89) mm, rotated rx 180 ry 0 rz 0.01 deg; joints [35.004, -36.023, 87.516, -138.456, 59.907, 156.991]
  MoveL 7360 to (-325.37, 265.7, -59.13) mm, rotated rx -180 ry 0 rz 0.01 deg; joints [35.076, -35.694, 86.832, -138.242, 59.671, 156.678]
  MoveL 7361 to (-331.81, 264.22, -59.37) mm, rotated rx -180 ry 0 rz 0.01 deg; joints [34.908, -35.453, 86.344, -138.323, 59.417, 156.58]
  MoveL 7362 to (-333.04, 257.73, -59.62) mm, rotated rx -180 ry 0 rz 0.01 deg; joints [34.701, -35.576, 86.638, -138.608, 59.458, 156.824]
  MoveL 7363 to (-327.58, 254.01, -59.86) mm, rotated rx -180 ry 0 rz 0.01 deg; joints [34.702, -35.901, 87.357, -138.759, 59.755, 157.125]
  MoveL 7364 to (-321.99, 257.51, -60.11) mm, rotated rx 180 ry 0 rz 0.01 deg; joints [34.912, -36.025, 87.638, -138.598, 59.959, 157.132]
  MoveL 7365 to (-322.95, 264.04, -60.35) mm, rotated rx 180 ry 0 rz 0.01 deg; joints [35.077, -35.787, 87.144, -138.326, 59.836, 156.846]
  MoveL 7366 to (-329.32, 265.78, -60.6) mm, rotated rx -180 ry 0 rz 0.01 deg; joints [35.001, -35.456, 86.462, -138.27, 59.541, 156.617]
  MoveL 7367 to (-333.47, 260.63, -60.84) mm, rotated rx -180 ry 0 rz 0.01 deg; joints [34.775, -35.418, 86.409, -138.503, 59.437, 156.73]
  MoveL 7368 to (-330.41, 254.78, -61.08) mm, rotated rx 180 ry 0 rz 0.01 deg; joints [34.669, -35.703, 87.048, -138.751, 59.658, 157.058]
  MoveL 7369 to (-323.82, 255.23, -61.33) mm, rotated rx 180 ry 0 rz 0.01 deg; joints [34.812, -35.956, 87.608, -138.719, 59.947, 157.215]
  MoveL 7370 to (-321.6, 261.45, -61.57) mm, rotated rx 180 ry 0 rz 0.01 deg; joints [35.031, -35.861, 87.418, -138.451, 59.967, 157.025]
  MoveL 7371 to (-326.4, 265.98, -61.82) mm, rotated rx -180 ry 0 rz 0.01 deg; joints [35.064, -35.517, 86.703, -138.273, 59.703, 156.722]
  MoveL 7372 to (-332.48, 263.39, -62.06) mm, rotated rx 180 ry 0 rz 0.01 deg; joints [34.872, -35.323, 86.317, -138.4, 59.479, 156.678]
  MoveL 7373 to (-332.54, 256.79, -62.3) mm, rotated rx -180 ry 0 rz 0.01 deg; joints [34.685, -35.498, 86.722, -138.688, 59.574, 156.957]
  MoveL 7374 to (-326.52, 254.08, -62.55) mm, rotated rx -180 ry 0 rz 0.01 deg; joints [34.727, -35.818, 87.429, -138.793, 59.882, 157.231]
  MoveL 7375 to (-321.63, 258.51, -62.79) mm, rotated rx 180 ry 0 rz 0.01 deg; joints [34.949, -35.886, 87.589, -138.594, 60.042, 157.181]
  MoveL 7376 to (-323.73, 264.78, -63.04) mm, rotated rx 180 ry 0 rz 0.01 deg; joints [35.084, -35.607, 87.01, -138.336, 59.873, 156.878]
  MoveL 7377 to (-330.31, 265.36, -63.28) mm, rotated rx 180 ry 0 rz 0.01 deg; joints [34.971, -35.302, 86.381, -138.33, 59.584, 156.69]
  MoveL 7378 to (-333.48, 259.57, -63.52) mm, rotated rx 180 ry 0 rz 0.01 deg; joints [34.746, -35.322, 86.456, -138.589, 59.531, 156.855]
  MoveL 7379 to (-329.44, 254.34, -63.77) mm, rotated rx -180 ry 0 rz 0.01 deg; joints [34.677, -35.631, 87.143, -138.807, 59.788, 157.182]
  MoveL 7380 to (-323.03, 255.94, -64.01) mm, rotated rx -180 ry 0 rz 0.01 deg; joints [34.849, -35.842, 87.615, -138.726, 60.053, 157.287]
  MoveL 7381 to (-321.94, 262.46, -64.26) mm, rotated rx -180 ry 0 rz 0.01 deg; joints [35.055, -35.691, 87.306, -138.449, 60.019, 157.056]
  MoveL 7382 to (-327.46, 266.07, -64.5) mm, rotated rx -180 ry 0 rz 0.01 deg; joints [35.047, -35.344, 86.583, -138.312, 59.735, 156.772]
  MoveL 7383 to (-327.82, 266.07, -64.5) mm, rotated rx 180 ry 0 rz 0.01 deg; joints [35.04, -35.329, 86.551, -138.312, 59.72, 156.762]
  MoveC 7384 to (-329.82, 265.24, -64.5) mm, rotated rx 180 ry 0 rz 0.01 deg; joints [34.977, -35.268, 86.423, -138.352, 59.643, 156.745] to (-330.66, 263.23, -64.5) mm, rotated rx 180 ry 0 rz 0.01 deg; joints [34.905, -35.291, 86.474, -138.44, 59.634, 156.806]
  MoveL 7385 to (-330.65, 221.91, -64.5) mm, rotated rx 180 ry 0 rz 0.01 deg; joints [33.726, -36.442, 88.995, -140.204, 60.199, 158.476]
  MoveC 7386 to (-329.57, 220.76, -64.5) mm, rotated rx -180 ry 0 rz 0.01 deg; joints [33.714, -36.518, 89.159, -140.25, 60.262, 158.548] to (-328.37, 221.79, -64.5) mm, rotated rx 180 ry 0 rz 0.01 deg; joints [33.767, -36.54, 89.205, -140.202, 60.3, 158.536]
  MoveL 7387 to (-324.25, 262.95, -64.5) mm, rotated rx 180 ry 0 rz 0.01 deg; joints [35.023, -35.569, 87.067, -138.437, 59.919, 156.984]
  MoveC 7388 to (-324.97, 265.14, -64.5) mm, rotated rx 180 ry 0 rz 0.01 deg; joints [35.07, -35.476, 86.866, -138.346, 59.857, 156.875] to (-327.07, 266.07, -64.5) mm, rotated rx 180 ry 0 rz 0.01 deg; joints [35.055, -35.361, 86.618, -138.311, 59.752, 156.782]
  MoveL 7389 to (-327.46, 266.07, -64.5) mm, rotated rx -180 ry 0 rz 0.01 deg; joints [35.047, -35.344, 86.583, -138.312, 59.735, 156.772]
  MoveC 7390 to (-329.64, 266.86, -64.5) mm, rotated rx 180 ry 0 rz 0.01 deg; joints [35.027, -35.229, 86.337, -138.282, 59.629, 156.682] to (-330.81, 268.87, -64.5) mm, rotated rx -180 ry 0 rz 0.01 deg; joints [35.06, -35.122, 86.105, -138.198, 59.55, 156.568]
  MoveC 7391 to (-332.54, 270.78, -64.5) mm, rotated rx 180 ry 0 rz 0.01 deg; joints [35.079, -34.992, 85.827, -138.12, 59.447, 156.442] to (-335.01, 270.03, -64.5) mm, rotated rx 180 ry 0 rz 0.01 deg; joints [35.01, -34.909, 85.65, -138.156, 59.349, 156.408]
  MoveC 7392 to (-335.71, 268.86, -64.5) mm, rotated rx 180 ry 0 rz 0.01 deg; joints [34.963, -34.913, 85.662, -138.208, 59.334, 156.439] to (-335.95, 267.51, -64.5) mm, rotated rx 180 ry 0 rz 0.01 deg; joints [34.921, -34.942, 85.725, -138.266, 59.342, 156.489]
  MoveL 7393 to (-335.95, 181.7, -64.5) mm, rotated rx -180 ry 0 rz 0.01 deg; joints [32.447, -37.275, 90.845, -141.93, 60.507, 159.899]
  MoveC 7394 to (-334.83, 179.88, -64.5) mm, rotated rx -180 ry 0 rz 0.01 deg; joints [32.414, -37.367, 91.046, -142.003, 60.58, 159.993] to (-332.7, 180.04, -64.5) mm, rotated rx 180 ry 0 rz 0.01 deg; joints [32.459, -37.451, 91.225, -141.988, 60.672, 160.037]
  MoveL 7395 to (-328.2, 183.28, -64.5) mm, rotated rx 180 ry 0 rz 0.01 deg; joints [32.641, -37.553, 91.44, -141.833, 60.826, 160.02]
  MoveC 7396 to (-327.12, 184.46, -64.5) mm, rotated rx 180 ry 0 rz 0.01 deg; joints [32.697, -37.567, 91.467, -141.779, 60.857, 160] to (-326.63, 185.99, -64.5) mm, rotated rx 180 ry 0 rz 0.01 deg; joints [32.751, -37.549, 91.425, -141.712, 60.859, 159.954]
  MoveL 7397 to (-318.46, 267.6, -64.5) mm, rotated rx 180 ry 0 rz 0.01 deg; joints [35.268, -35.678, 87.292, -138.224, 60.107, 156.941]
  MoveC 7398 to (-319.33, 270.24, -64.5) mm, rotated rx 180 ry 0 rz 0.01 deg; joints [35.325, -35.566, 87.048, -138.114, 60.033, 156.81] to (-321.87, 271.37, -64.5) mm, rotated rx 180 ry 0 rz 0.01 deg; joints [35.306, -35.427, 86.751, -138.072, 59.907, 156.698]
  MoveL 7399 to (-332.1, 271.37, -64.5) mm, rotated rx -180 ry 0 rz 0.01 deg; joints [35.104, -34.994, 85.83, -138.094, 59.459, 156.429]
  MoveC 7400 to (-333.7, 271.02, -64.5) mm, rotated rx 180 ry 0 rz 0.01 deg; joints [35.063, -34.936, 85.707, -138.112, 59.393, 156.401] to (-335.01, 270.03, -64.5) mm, rotated rx -180 ry 0 rz 0.01 deg; joints [35.01, -34.909, 85.65, -138.156, 59.349, 156.408]
  MoveC 7401 to (-337.39, 267.84, -64.5) mm, rotated rx 180 ry 0 rz 0.01 deg; joints [34.902, -34.871, 85.573, -138.254, 59.274, 156.437] to (-340.21, 266.23, -64.5) mm, rotated rx -180 ry 0 rz 0.01 deg; joints [34.802, -34.797, 85.418, -138.328, 59.171, 156.429]
  MoveC 7402 to (-342.79, 264.08, -64.5) mm, rotated rx -180 ry 0 rz 0.01 deg; joints [34.692, -34.748, 85.318, -138.424, 59.086, 156.45] to (-343.76, 260.86, -64.5) mm, rotated rx -180 ry 0 rz 0.01 deg; joints [34.583, -34.8, 85.433, -138.564, 59.087, 156.559]
  MoveL 7403 to (-343.76, 166.47, -64.5) mm, rotated rx -180 ry 0 rz 0.01 deg; joints [31.848, -37.335, 90.999, -142.605, 60.364, 160.289]
  MoveC 7404 to (-342.64, 164.65, -64.5) mm, rotated rx 180 ry 0 rz 0.01 deg; joints [31.814, -37.427, 91.199, -142.679, 60.437, 160.382] to (-340.51, 164.81, -64.5) mm, rotated rx -180 ry 0 rz 0.01 deg; joints [31.858, -37.511, 91.379, -142.664, 60.53, 160.425]
  MoveL 7405 to (-323.84, 176.79, -64.5) mm, rotated rx 180 ry 0 rz 0.01 deg; joints [32.531, -37.894, 92.183, -142.089, 61.103, 160.361]
  MoveC 7406 to (-320.41, 180.58, -64.5) mm, rotated rx 180 ry 0 rz 0.01 deg; joints [32.71, -37.938, 92.271, -141.913, 61.202, 160.299] to (-318.84, 185.45, -64.5) mm, rotated rx -180 ry 0 rz 0.01 deg; joints [32.885, -37.879, 92.135, -141.701, 61.206, 160.153]
  MoveL 7407 to (-309.83, 275.41, -64.5) mm, rotated rx -180 ry 0 rz 0.01 deg; joints [35.66, -35.811, 87.564, -137.866, 60.373, 156.84]
  MoveC 7408 to (-310.7, 278.05, -64.5) mm, rotated rx -180 ry 0 rz 0.01 deg; joints [35.717, -35.699, 87.32, -137.757, 60.299, 156.709] to (-313.24, 279.18, -64.5) mm, rotated rx -180 ry 0 rz 0.01 deg; joints [35.697, -35.561, 87.024, -137.716, 60.174, 156.597]
  MoveL 7409 to (-339.91, 279.17, -64.5) mm, rotated rx 180 ry 0 rz 0.01 deg; joints [35.169, -34.43, 84.618, -137.768, 59.005, 155.889]
  MoveC 7410 to (-342.63, 278.05, -64.5) mm, rotated rx -180 ry 0 rz 0.01 deg; joints [35.084, -34.345, 84.441, -137.819, 58.9, 155.863] to (-343.76, 275.32, -64.5) mm, rotated rx -180 ry 0 rz 0.01 deg; joints [34.987, -34.377, 84.512, -137.938, 58.888, 155.948]
  MoveL 7411 to (-343.76, 260.86, -64.5) mm, rotated rx 180 ry 0 rz 0.01 deg; joints [34.583, -34.8, 85.433, -138.564, 59.087, 156.559]
  MoveC 7412 to (-344.82, 257.34, -64.5) mm, rotated rx 180 ry 0 rz 0.01 deg; joints [34.463, -34.856, 85.557, -138.718, 59.088, 156.678] to (-347.66, 255, -64.5) mm, rotated rx -180 ry 0 rz 0.01 deg; joints [34.343, -34.801, 85.443, -138.822, 58.994, 156.7]
  MoveC 7413 to (-350.5, 252.67, -64.5) mm, rotated rx 180 ry 0 rz 0.01 deg; joints [34.222, -34.745, 85.328, -138.926, 58.899, 156.722] to (-351.57, 249.15, -64.5) mm, rotated rx -180 ry 0 rz 0.01 deg; joints [34.103, -34.799, 85.449, -139.08, 58.9, 156.84]
  MoveL 7414 to (-351.57, 151.24, -64.5) mm, rotated rx 180 ry 0 rz 0.01 deg; joints [31.247, -37.387, 91.135, -143.28, 60.217, 160.674]
  MoveC 7415 to (-350.45, 149.42, -64.5) mm, rotated rx -180 ry 0 rz 0.01 deg; joints [31.213, -37.477, 91.333, -143.354, 60.29, 160.766] to (-348.32, 149.58, -64.5) mm, rotated rx -180 ry 0 rz 0.01 deg; joints [31.256, -37.562, 91.514, -143.34, 60.383, 160.809]
  MoveL 7416 to (-316.69, 172.31, -64.5) mm, rotated rx 180 ry 0 rz 0.01 deg; joints [32.533, -38.295, 93.052, -142.243, 61.474, 160.688]
  MoveC 7417 to (-313.05, 176.33, -64.5) mm, rotated rx 180 ry 0 rz 0.01 deg; joints [32.724, -38.341, 93.144, -142.056, 61.578, 160.621] to (-311.39, 181.5, -64.5) mm, rotated rx 180 ry 0 rz 0.01 deg; joints [32.91, -38.278, 93.001, -141.831, 61.581, 160.469]
  MoveL 7418 to (-301.2, 283.22, -64.5) mm, rotated rx 180 ry 0 rz 0.01 deg; joints [36.053, -35.94, 87.828, -137.507, 60.636, 156.738]
  MoveC 7419 to (-302.07, 285.86, -64.5) mm, rotated rx 180 ry 0 rz 0.01 deg; joints [36.109, -35.828, 87.583, -137.398, 60.562, 156.606] to (-304.61, 286.99, -64.5) mm, rotated rx 180 ry 0 rz 0.01 deg; joints [36.089, -35.69, 87.288, -137.359, 60.438, 156.495]
  MoveL 7420 to (-347.72, 286.98, -64.5) mm, rotated rx 180 ry 0 rz 0.01 deg; joints [35.232, -33.856, 83.389, -137.433, 58.549, 155.337]
  MoveC 7421 to (-350.44, 285.86, -64.5) mm, rotated rx 180 ry 0 rz 0.01 deg; joints [35.148, -33.771, 83.209, -137.482, 58.443, 155.309] to (-351.57, 283.13, -64.5) mm, rotated rx 180 ry 0 rz 0.01 deg; joints [35.051, -33.803, 83.282, -137.601, 58.43, 155.396]
  MoveL 7422 to (-351.57, 249.15, -64.5) mm, rotated rx 180 ry 0 rz 0.01 deg; joints [34.103, -34.799, 85.449, -139.08, 58.9, 156.84]
  MoveC 7423 to (-352.63, 245.63, -64.5) mm, rotated rx 180 ry 0 rz 0.01 deg; joints [33.983, -34.853, 85.57, -139.233, 58.9, 156.957] to (-355.47, 243.29, -64.5) mm, rotated rx -180 ry 0 rz 0.01 deg; joints [33.863, -34.797, 85.453, -139.337, 58.805, 156.979]
  MoveC 7424 to (-358.31, 240.95, -64.5) mm, rotated rx 180 ry 0 rz 0.01 deg; joints [33.743, -34.74, 85.335, -139.441, 58.709, 157] to (-359.38, 237.43, -64.5) mm, rotated rx -180 ry 0 rz 0.01 deg; joints [33.623, -34.792, 85.453, -139.595, 58.709, 157.117]
  MoveL 7425 to (-359.38, 136.01, -64.5) mm, rotated rx 180 ry 0 rz 0.01 deg; joints [30.646, -37.429, 91.252, -143.955, 60.066, 161.055]
  MoveC 7426 to (-358.26, 134.19, -64.5) mm, rotated rx 180 ry 0 rz 0.01 deg; joints [30.611, -37.519, 91.448, -144.029, 60.14, 161.146] to (-356.13, 134.35, -64.5) mm, rotated rx 180 ry 0 rz 0.01 deg; joints [30.654, -37.604, 91.631, -144.015, 60.233, 161.188]
  MoveL 7427 to (-309.27, 168.03, -64.5) mm, rotated rx 180 ry 0 rz 0.01 deg; joints [32.547, -38.697, 93.926, -142.384, 61.852, 161.008]
  MoveC 7428 to (-305.63, 172.05, -64.5) mm, rotated rx -180 ry 0 rz 0.01 deg; joints [32.738, -38.742, 94.017, -142.196, 61.956, 160.942] to (-303.97, 177.21, -64.5) mm, rotated rx -180 ry 0 rz 0.01 deg; joints [32.926, -38.68, 93.875, -141.971, 61.958, 160.791]
  MoveL 7429 to (-292.57, 291.03, -64.5) mm, rotated rx 180 ry 0 rz 0.01 deg; joints [36.448, -36.065, 88.082, -137.145, 60.896, 156.634]
  MoveC 7430 to (-293.44, 293.67, -64.5) mm, rotated rx -180 ry 0 rz 0.01 deg; joints [36.503, -35.952, 87.837, -137.038, 60.822, 156.502] to (-295.97, 294.8, -64.5) mm, rotated rx 180 ry 0 rz 0.01 deg; joints [36.482, -35.815, 87.543, -136.999, 60.699, 156.391]
  MoveL 7431 to (-355.53, 294.79, -64.5) mm, rotated rx -180 ry 0 rz 0.01 deg; joints [35.295, -33.273, 82.141, -137.088, 58.089, 154.772]
  MoveC 7432 to (-358.25, 293.67, -64.5) mm, rotated rx -180 ry 0 rz 0.01 deg; joints [35.212, -33.186, 81.959, -137.136, 57.982, 154.743] to (-359.38, 290.94, -64.5) mm, rotated rx -180 ry 0 rz 0.01 deg; joints [35.115, -33.219, 82.034, -137.255, 57.969, 154.831]
  MoveL 7433 to (-359.38, 237.43, -64.5) mm, rotated rx 180 ry 0 rz 0.01 deg; joints [33.623, -34.792, 85.453, -139.595, 58.709, 157.117]
  MoveC 7434 to (-360.44, 233.91, -64.5) mm, rotated rx 180 ry 0 rz 0.01 deg; joints [33.502, -34.845, 85.57, -139.749, 58.709, 157.234] to (-363.28, 231.57, -64.5) mm, rotated rx -180 ry 0 rz 0.01 deg; joints [33.382, -34.787, 85.449, -139.852, 58.613, 157.255]
  MoveC 7435 to (-366.12, 229.24, -64.5) mm, rotated rx -180 ry 0 rz 0.01 deg; joints [33.263, -34.728, 85.328, -139.956, 58.516, 157.276] to (-367.19, 225.72, -64.5) mm, rotated rx -180 ry 0 rz 0.01 deg; joints [33.142, -34.779, 85.443, -140.11, 58.516, 157.392]
  MoveL 7436 to (-367.18, 120.78, -64.5) mm, rotated rx 180 ry 0 rz 0.01 deg; joints [30.044, -37.462, 91.35, -144.63, 59.911, 161.431]
  MoveC 7437 to (-366.07, 118.96, -64.5) mm, rotated rx 180 ry 0 rz 0.01 deg; joints [30.008, -37.552, 91.545, -144.704, 59.985, 161.522] to (-363.94, 119.12, -64.5) mm, rotated rx 180 ry 0 rz 0.01 deg; joints [30.05, -37.637, 91.728, -144.691, 60.079, 161.564]
  MoveL 7438 to (-301.85, 163.74, -64.5) mm, rotated rx -180 ry 0 rz 0.01 deg; joints [32.561, -39.095, 94.792, -142.521, 62.229, 161.325]
  MoveC 7439 to (-298.21, 167.76, -64.5) mm, rotated rx 180 ry 0 rz 0.01 deg; joints [32.753, -39.14, 94.883, -142.332, 62.331, 161.259] to (-296.55, 172.93, -64.5) mm, rotated rx 180 ry 0 rz 0.01 deg; joints [32.942, -39.079, 94.742, -142.106, 62.333, 161.109]
  MoveL 7440 to (-283.94, 298.84, -64.5) mm, rotated rx -180 ry 0 rz 0.01 deg; joints [36.843, -36.185, 88.327, -136.782, 61.153, 156.528]
  MoveC 7441 to (-284.81, 301.48, -64.5) mm, rotated rx 180 ry 0 rz 0.01 deg; joints [36.898, -36.072, 88.081, -136.675, 61.079, 156.397] to (-287.34, 302.61, -64.5) mm, rotated rx 180 ry 0 rz 0.01 deg; joints [36.876, -35.936, 87.789, -136.638, 60.957, 156.285]
  MoveL 7442 to (-363.34, 302.6, -64.5) mm, rotated rx -180 ry 0 rz 0.01 deg; joints [35.357, -32.679, 80.875, -136.734, 57.625, 154.193]
  MoveC 7443 to (-366.06, 301.47, -64.5) mm, rotated rx 180 ry 0 rz 0.01 deg; joints [35.274, -32.591, 80.69, -136.78, 57.517, 154.162] to (-367.19, 298.75, -64.5) mm, rotated rx -180 ry 0 rz 0.01 deg; joints [35.178, -32.625, 80.766, -136.899, 57.504, 154.252]
  MoveL 7444 to (-367.19, 225.72, -64.5) mm, rotated rx 180 ry 0 rz 0.01 deg; joints [33.142, -34.779, 85.443, -140.11, 58.516, 157.392]
  MoveC 7445 to (-368.25, 222.2, -64.5) mm, rotated rx -180 ry 0 rz 0.01 deg; joints [33.022, -34.83, 85.557, -140.263, 58.515, 157.508] to (-371.09, 219.86, -64.5) mm, rotated rx 180 ry 0 rz 0.01 deg; joints [32.902, -34.77, 85.433, -140.367, 58.418, 157.529]
  MoveC 7446 to (-373.93, 217.52, -64.5) mm, rotated rx 180 ry 0 rz 0.01 deg; joints [32.783, -34.71, 85.308, -140.47, 58.32, 157.549] to (-375, 214, -64.5) mm, rotated rx -180 ry 0 rz 0.01 deg; joints [32.662, -34.76, 85.42, -140.624, 58.319, 157.665]
  MoveL 7447 to (-374.99, 105.55, -64.5) mm, rotated rx 180 ry 0 rz 0.01 deg; joints [29.441, -37.487, 91.429, -145.304, 59.752, 161.804]
  MoveC 7448 to (-373.88, 103.73, -64.5) mm, rotated rx 180 ry 0 rz 0.01 deg; joints [29.404, -37.576, 91.623, -145.379, 59.826, 161.893] to (-371.75, 103.89, -64.5) mm, rotated rx 180 ry 0 rz 0.01 deg; joints [29.446, -37.662, 91.807, -145.366, 59.921, 161.935]
  MoveL 7449 to (-293.62, 160.04, -64.5) mm, rotated rx 180 ry 0 rz 0.01 deg; joints [32.608, -39.506, 95.688, -142.625, 62.63, 161.633]
  MoveC 7450 to (-290.6, 163.37, -64.5) mm, rotated rx 180 ry 0 rz 0.01 deg; joints [32.768, -39.543, 95.762, -142.467, 62.714, 161.579] to (-289.22, 167.65, -64.5) mm, rotated rx -180 ry 0 rz 0.01 deg; joints [32.926, -39.493, 95.646, -142.28, 62.715, 161.456]
  MoveL 7451 to (-275.69, 303.58, -64.5) mm, rotated rx -180 ry 0 rz 0.01 deg; joints [37.146, -36.376, 88.728, -136.547, 61.433, 156.539]
  MoveC 7452 to (-275.56, 304.4, -64.5) mm, rotated rx -180 ry 0 rz 0.01 deg; joints [37.172, -36.357, 88.686, -136.513, 61.427, 156.508] to (-275.41, 305.21, -64.5) mm, rotated rx 180 ry 0 rz 0.01 deg; joints [37.197, -36.339, 88.647, -136.478, 61.422, 156.478]
  MoveC 7453 to (-275.26, 306.02, -64.5) mm, rotated rx 180 ry 0 rz 0.01 deg; joints [37.223, -36.321, 88.607, -136.444, 61.417, 156.448] to (-275.12, 306.84, -64.5) mm, rotated rx 180 ry 0 rz 0.01 deg; joints [37.248, -36.303, 88.566, -136.409, 61.412, 156.418]
  MoveC 7454 to (-275.84, 309.33, -64.5) mm, rotated rx 180 ry 0 rz 0.01 deg; joints [37.302, -36.2, 88.343, -136.308, 61.347, 156.296] to (-278.19, 310.42, -64.5) mm, rotated rx 180 ry 0 rz 0.01 deg; joints [37.282, -36.073, 88.07, -136.273, 61.233, 156.191]
  MoveL 7455 to (-371.15, 310.41, -64.5) mm, rotated rx 180 ry 0 rz 0.01 deg; joints [35.418, -32.075, 79.587, -136.369, 57.158, 153.6]
  MoveC 7456 to (-373.87, 309.28, -64.5) mm, rotated rx 180 ry 0 rz 0.01 deg; joints [35.336, -31.986, 79.4, -136.413, 57.048, 153.568] to (-375, 306.56, -64.5) mm, rotated rx -180 ry 0 rz 0.01 deg; joints [35.241, -32.021, 79.478, -136.532, 57.035, 153.658]
  MoveL 7457 to (-375, 214, -64.5) mm, rotated rx 180 ry 0 rz 0.01 deg; joints [32.662, -34.76, 85.42, -140.624, 58.319, 157.665]
  MoveC 7458 to (-376.06, 210.48, -64.5) mm, rotated rx -180 ry 0 rz 0.01 deg; joints [32.542, -34.809, 85.531, -140.777, 58.318, 157.78] to (-378.9, 208.14, -64.5) mm, rotated rx 180 ry 0 rz 0.01 deg; joints [32.422, -34.748, 85.404, -140.88, 58.219, 157.8]
  MoveC 7459 to (-381.74, 205.81, -64.5) mm, rotated rx -180 ry 0 rz 0.01 deg; joints [32.303, -34.686, 85.276, -140.983, 58.12, 157.82] to (-382.81, 202.29, -64.5) mm, rotated rx -180 ry 0 rz 0.01 deg; joints [32.183, -34.734, 85.384, -141.137, 58.119, 157.935]
  MoveL 7460 to (-382.8, 90.32, -64.5) mm, rotated rx 180 ry 0 rz 0.01 deg; joints [28.837, -37.502, 91.489, -145.978, 59.588, 162.172]
  MoveC 7461 to (-381.69, 88.5, -64.5) mm, rotated rx -180 ry 0 rz 0.01 deg; joints [28.8, -37.591, 91.681, -146.053, 59.662, 162.261] to (-379.56, 88.66, -64.5) mm, rotated rx -180 ry 0 rz 0.01 deg; joints [28.841, -37.677, 91.867, -146.041, 59.758, 162.302]
  MoveL 7462 to (-288.34, 154.36, -64.5) mm, rotated rx -180 ry 0 rz 0.01 deg; joints [32.537, -39.846, 96.435, -142.827, 62.93, 161.945]
  MoveC 7463 to (-287.56, 154.88, -64.5) mm, rotated rx 180 ry 0 rz 0.01 deg; joints [32.569, -39.864, 96.473, -142.799, 62.956, 161.943] to (-286.73, 155.35, -64.5) mm, rotated rx 180 ry 0 rz 0.01 deg; joints [32.599, -39.885, 96.517, -142.774, 62.985, 161.944]
  MoveC 7464 to (-285.89, 155.79, -64.5) mm, rotated rx 180 ry 0 rz 0.01 deg; joints [32.629, -39.907, 96.564, -142.75, 63.015, 161.946] to (-285.05, 156.22, -64.5) mm, rotated rx 180 ry 0 rz 0.01 deg; joints [32.659, -39.929, 96.611, -142.727, 63.045, 161.949]
  MoveC 7465 to (-282.42, 158.72, -64.5) mm, rotated rx 180 ry 0 rz 0.01 deg; joints [32.787, -39.971, 96.697, -142.605, 63.122, 161.916] to (-281.6, 162.25, -64.5) mm, rotated rx -180 ry 0 rz 0.01 deg; joints [32.911, -39.918, 96.576, -142.452, 63.11, 161.809]
  MoveC 7466 to (-281.65, 163.23, -64.5) mm, rotated rx -180 ry 0 rz 0.01 deg; joints [32.94, -39.892, 96.518, -142.412, 63.094, 161.773] to (-281.7, 164.22, -64.5) mm, rotated rx 180 ry 0 rz 0.01 deg; joints [32.97, -39.866, 96.461, -142.371, 63.079, 161.737]
  MoveC 7467 to (-281.71, 165.21, -64.5) mm, rotated rx -180 ry 0 rz 0.01 deg; joints [33, -39.842, 96.407, -142.33, 63.066, 161.702] to (-281.65, 166.2, -64.5) mm, rotated rx 180 ry 0 rz 0.01 deg; joints [33.031, -39.821, 96.359, -142.289, 63.055, 161.668]
  MoveL 7468 to (-267.34, 307.3, -64.5) mm, rotated rx -180 ry 0 rz 0.01 deg; joints [37.425, -36.599, 89.198, -136.352, 61.729, 156.593]
  MoveC 7469 to (-266.87, 309.19, -64.5) mm, rotated rx 180 ry 0 rz 0.01 deg; joints [37.487, -36.562, 89.116, -136.271, 61.723, 156.526] to (-266.31, 311.05, -64.5) mm, rotated rx 180 ry 0 rz 0.01 deg; joints [37.55, -36.528, 89.042, -136.191, 61.72, 156.463]
  MoveC 7470 to (-265.72, 312.9, -64.5) mm, rotated rx 180 ry 0 rz 0.01 deg; joints [37.614, -36.497, 88.972, -136.111, 61.719, 156.401] to (-265.16, 314.76, -64.5) mm, rotated rx 180 ry 0 rz 0.01 deg; joints [37.677, -36.464, 88.898, -136.031, 61.717, 156.337]
  MoveC 7471 to (-265.58, 317.14, -64.5) mm, rotated rx 180 ry 0 rz 0.01 deg; joints [37.733, -36.376, 88.706, -135.935, 61.666, 156.227] to (-267.75, 318.23, -64.5) mm, rotated rx -180 ry 0 rz 0.01 deg; joints [37.717, -36.257, 88.452, -135.9, 61.561, 156.128]
  MoveL 7472 to (-378.96, 318.22, -64.5) mm, rotated rx 180 ry 0 rz 0.01 deg; joints [35.479, -31.46, 78.279, -135.993, 56.686, 152.992]
  MoveC 7473 to (-381.68, 317.09, -64.5) mm, rotated rx 180 ry 0 rz 0.01 deg; joints [35.397, -31.369, 78.089, -136.034, 56.575, 152.958] to (-382.81, 314.37, -64.5) mm, rotated rx 180 ry 0 rz 0.01 deg; joints [35.302, -31.405, 78.168, -136.154, 56.562, 153.05]
  MoveL 7474 to (-382.81, 202.29, -64.5) mm, rotated rx 180 ry 0 rz 0.01 deg; joints [32.183, -34.734, 85.384, -141.137, 58.119, 157.935]
  MoveC 7475 to (-383.87, 198.77, -64.5) mm, rotated rx 180 ry 0 rz 0.01 deg; joints [32.062, -34.782, 85.491, -141.291, 58.117, 158.049] to (-386.71, 196.43, -64.5) mm, rotated rx -180 ry 0 rz 0.01 deg; joints [31.943, -34.719, 85.361, -141.393, 58.018, 158.069]
  MoveC 7476 to (-389.55, 194.09, -64.5) mm, rotated rx 180 ry 0 rz 0.01 deg; joints [31.824, -34.656, 85.23, -141.495, 57.918, 158.089] to (-390.62, 190.57, -64.5) mm, rotated rx 180 ry 0 rz 0.01 deg; joints [31.703, -34.702, 85.335, -141.649, 57.916, 158.202]
  MoveL 7477 to (-390.61, 75.09, -64.5) mm, rotated rx -180 ry 0 rz 0.01 deg; joints [28.234, -37.509, 91.53, -146.652, 59.42, 162.537]
  MoveC 7478 to (-389.5, 73.27, -64.5) mm, rotated rx -180 ry 0 rz 0.01 deg; joints [28.195, -37.597, 91.721, -146.727, 59.494, 162.625] to (-387.37, 73.43, -64.5) mm, rotated rx -180 ry 0 rz 0.01 deg; joints [28.236, -37.684, 91.909, -146.715, 59.591, 162.666]
  MoveL 7479 to (-283.89, 148.16, -64.5) mm, rotated rx 180 ry 0 rz 0.01 deg; joints [32.434, -40.164, 97.135, -143.053, 63.201, 162.255]
  MoveC 7480 to (-281.83, 149.43, -64.5) mm, rotated rx 180 ry 0 rz 0.01 deg; joints [32.513, -40.213, 97.24, -142.986, 63.271, 162.253] to (-279.6, 150.38, -64.5) mm, rotated rx -180 ry 0 rz 0.01 deg; joints [32.587, -40.276, 97.375, -142.93, 63.353, 162.266]
  MoveC 7481 to (-277.29, 151.09, -64.5) mm, rotated rx 180 ry 0 rz 0.01 deg; joints [32.654, -40.347, 97.529, -142.884, 63.44, 162.289] to (-274.94, 151.66, -64.5) mm, rotated rx 180 ry 0 rz 0.01 deg; joints [32.718, -40.423, 97.693, -142.843, 63.532, 162.318]
  MoveC 7482 to (-272.9, 153.12, -64.5) mm, rotated rx 180 ry 0 rz 0.01 deg; joints [32.804, -40.467, 97.784, -142.767, 63.598, 162.309] to (-272.61, 155.62, -64.5) mm, rotated rx -180 ry 0 rz 0.01 deg; joints [32.886, -40.419, 97.676, -142.661, 63.577, 162.228]
  MoveC 7483 to (-273.09, 157.3, -64.5) mm, rotated rx -180 ry 0 rz 0.01 deg; joints [32.929, -40.361, 97.546, -142.595, 63.534, 162.16] to (-273.5, 159.01, -64.5) mm, rotated rx 180 ry 0 rz 0.01 deg; joints [32.973, -40.305, 97.421, -142.528, 63.494, 162.092]
  MoveC 7484 to (-273.81, 160.74, -64.5) mm, rotated rx 180 ry 0 rz 0.01 deg; joints [33.02, -40.251, 97.303, -142.459, 63.458, 162.025] to (-274, 162.48, -64.5) mm, rotated rx 180 ry 0 rz 0.01 deg; joints [33.069, -40.202, 97.194, -142.388, 63.426, 161.96]
  MoveC 7485 to (-274.06, 163.22, -64.5) mm, rotated rx -180 ry 0 rz 0.01 deg; joints [33.091, -40.183, 97.15, -142.358, 63.414, 161.933] to (-274.1, 163.96, -64.5) mm, rotated rx 180 ry 0 rz 0.01 deg; joints [33.113, -40.163, 97.106, -142.327, 63.403, 161.906]
  MoveC 7486 to (-274.11, 164.7, -64.5) mm, rotated rx -180 ry 0 rz 0.01 deg; joints [33.135, -40.145, 97.066, -142.297, 63.392, 161.88] to (-274.06, 165.44, -64.5) mm, rotated rx 180 ry 0 rz 0.01 deg; joints [33.159, -40.129, 97.03, -142.266, 63.384, 161.854]
  MoveL 7487 to (-260.01, 305.68, -64.5) mm, rotated rx -180 ry 0 rz 0.01 deg; joints [37.536, -36.936, 89.922, -136.381, 62.055, 156.84]
  MoveC 7488 to (-259.13, 309.22, -64.5) mm, rotated rx 180 ry 0 rz 0.01 deg; joints [37.652, -36.866, 89.768, -136.229, 62.043, 156.716] to (-258.06, 312.71, -64.5) mm, rotated rx 180 ry 0 rz 0.01 deg; joints [37.772, -36.805, 89.631, -136.079, 62.038, 156.598]
  MoveC 7489 to (-256.74, 316.11, -64.5) mm, rotated rx 180 ry 0 rz 0.01 deg; joints [37.894, -36.756, 89.521, -135.931, 62.046, 156.49] to (-255.08, 319.36, -64.5) mm, rotated rx 180 ry 0 rz 0.01 deg; joints [38.019, -36.724, 89.448, -135.788, 62.069, 156.396]
  MoveC 7490 to (-254.57, 320.2, -64.5) mm, rotated rx -180 ry 0 rz 0.01 deg; joints [38.053, -36.718, 89.435, -135.75, 62.078, 156.374] to (-254.05, 321.02, -64.5) mm, rotated rx -180 ry 0 rz 0.01 deg; joints [38.087, -36.714, 89.425, -135.713, 62.088, 156.353]
  MoveC 7491 to (-253.52, 321.85, -64.5) mm, rotated rx 180 ry 0 rz 0.01 deg; joints [38.12, -36.71, 89.415, -135.676, 62.098, 156.331] to (-253.02, 322.69, -64.5) mm, rotated rx -180 ry 0 rz 0.01 deg; joints [38.154, -36.705, 89.402, -135.639, 62.107, 156.309]
  MoveC 7492 to (-253.02, 324.92, -64.5) mm, rotated rx 180 ry 0 rz 0.01 deg; joints [38.215, -36.638, 89.255, -135.547, 62.076, 156.216] to (-254.95, 326.04, -64.5) mm, rotated rx 180 ry 0 rz 0.01 deg; joints [38.204, -36.528, 89.019, -135.511, 61.981, 156.121]
  MoveL 7493 to (-386.77, 326.03, -64.5) mm, rotated rx 180 ry 0 rz 0.01 deg; joints [35.539, -30.833, 76.948, -135.604, 56.21, 152.367]
  MoveC 7494 to (-389.49, 324.9, -64.5) mm, rotated rx 180 ry 0 rz 0.01 deg; joints [35.457, -30.74, 76.755, -135.643, 56.098, 152.331] to (-390.62, 322.18, -64.5) mm, rotated rx 180 ry 0 rz 0.01 deg; joints [35.363, -30.777, 76.836, -135.763, 56.084, 152.425]
  MoveL 7495 to (-390.62, 190.57, -64.5) mm, rotated rx 180 ry 0 rz 0.01 deg; joints [31.703, -34.702, 85.335, -141.649, 57.916, 158.202]
  MoveC 7496 to (-391.68, 187.05, -64.5) mm, rotated rx -180 ry 0 rz 0.01 deg; joints [31.582, -34.749, 85.439, -141.803, 57.913, 158.316] to (-394.52, 184.71, -64.5) mm, rotated rx 180 ry 0 rz 0.01 deg; joints [31.463, -34.684, 85.305, -141.905, 57.813, 158.335]
  MoveC 7497 to (-397.36, 182.38, -64.5) mm, rotated rx -180 ry 0 rz 0.01 deg; joints [31.345, -34.619, 85.171, -142.007, 57.712, 158.355] to (-398.43, 178.86, -64.5) mm, rotated rx -180 ry 0 rz 0.01 deg; joints [31.223, -34.664, 85.273, -142.161, 57.709, 158.468]
  MoveL 7498 to (-398.42, 58.56, -64.5) mm, rotated rx 180 ry 0 rz 0.01 deg; joints [27.589, -37.535, 91.615, -147.381, 59.263, 162.943]
  MoveC 7499 to (-397.35, 56.92, -64.5) mm, rotated rx -180 ry 0 rz 0.01 deg; joints [27.555, -37.616, 91.793, -147.449, 59.334, 163.023] to (-395.41, 57.25, -64.5) mm, rotated rx 180 ry 0 rz 0.01 deg; joints [27.597, -37.692, 91.955, -147.431, 59.42, 163.053]
  MoveC 7500 to (-393.89, 58.67, -64.5) mm, rotated rx 180 ry 0 rz 0.01 deg; joints [27.667, -37.726, 92.026, -147.365, 59.473, 163.037] to (-392.4, 60.12, -64.5) mm, rotated rx 180 ry 0 rz 0.01 deg; joints [27.737, -37.759, 92.094, -147.299, 59.525, 163.019]
  MoveC 7501 to (-390.85, 61.53, -64.5) mm, rotated rx 180 ry 0 rz 0.01 deg; joints [27.806, -37.794, 92.168, -147.235, 59.579, 163.003] to (-389.21, 62.81, -64.5) mm, rotated rx -180 ry 0 rz 0.01 deg; joints [27.874, -37.837, 92.256, -147.176, 59.639, 162.994]
  MoveL 7502 to (-279.48, 142.02, -64.5) mm, rotated rx 180 ry 0 rz 0.01 deg; joints [32.331, -40.477, 97.825, -143.276, 63.469, 162.558]
  MoveC 7503 to (-274.51, 144.37, -64.5) mm, rotated rx 180 ry 0 rz 0.01 deg; joints [32.501, -40.61, 98.112, -143.141, 63.647, 162.578] to (-269.04, 144.82, -64.5) mm, rotated rx 180 ry 0 rz 0.01 deg; joints [32.624, -40.807, 98.539, -143.08, 63.87, 162.674]
  MoveC 7504 to (-263.7, 143.92, -64.5) mm, rotated rx 180 ry 0 rz 0.01 deg; joints [32.702, -41.028, 99.023, -143.075, 64.105, 162.812] to (-258.52, 142.31, -64.5) mm, rotated rx 180 ry 0 rz 0.01 deg; joints [32.756, -41.259, 99.528, -143.098, 64.342, 162.97]
  MoveC 7505 to (-257.67, 141.96, -64.5) mm, rotated rx 180 ry 0 rz 0.01 deg; joints [32.762, -41.299, 99.616, -143.105, 64.382, 163] to (-256.83, 141.55, -64.5) mm, rotated rx 180 ry 0 rz 0.01 deg; joints [32.766, -41.339, 99.705, -143.115, 64.423, 163.03]
  MoveC 7506 to (-256.01, 141.12, -64.5) mm, rotated rx -180 ry 0 rz 0.01 deg; joints [32.769, -41.379, 99.794, -143.126, 64.462, 163.061] to (-255.2, 140.67, -64.5) mm, rotated rx 180 ry 0 rz 0.01 deg; joints [32.771, -41.42, 99.883, -143.137, 64.502, 163.092]
  MoveL 7507 to (-219.43, 120.08, -64.5) mm, rotated rx 180 ry 0 rz 0.01 deg; joints [32.85, -43.179, 103.782, -143.64, 66.243, 164.46]
  MoveC 7508 to (-215.28, 116.09, -64.5) mm, rotated rx 180 ry 0 rz 0.01 deg; joints [32.807, -43.414, 104.306, -143.759, 66.465, 164.666] to (-213.46, 110.64, -64.5) mm, rotated rx -180 ry 0 rz 0.01 deg; joints [32.669, -43.596, 104.72, -143.963, 66.612, 164.874]
  MoveC 7509 to (-214.2, 104.97, -64.5) mm, rotated rx 180 ry 0 rz 0.01 deg; joints [32.47, -43.692, 104.944, -144.203, 66.659, 165.04] to (-217.18, 100.1, -64.5) mm, rotated rx 180 ry 0 rz 0.01 deg; joints [32.249, -43.692, 104.951, -144.436, 66.604, 165.139]
  MoveC 7510 to (-218.18, 99.19, -64.5) mm, rotated rx -180 ry 0 rz 0.01 deg; joints [32.199, -43.676, 104.918, -144.484, 66.576, 165.149] to (-219.3, 98.44, -64.5) mm, rotated rx -180 ry 0 rz 0.01 deg; joints [32.152, -43.653, 104.868, -144.527, 66.54, 165.153]
  MoveL 7511 to (-328.52, 36.08, -64.5) mm, rotated rx -180 ry 0 rz 0.01 deg; joints [28.049, -40.869, 98.875, -148.042, 62.72, 165.093]
  MoveC 7512 to (-329.5, 34.8, -64.5) mm, rotated rx -180 ry 0 rz 0.01 deg; joints [27.99, -40.856, 98.849, -148.102, 62.693, 165.115] to (-329.29, 33.19, -64.5) mm, rotated rx 180 ry 0 rz 0.01 deg; joints [27.941, -40.896, 98.94, -148.168, 62.722, 165.17]
  MoveL 7513 to (-328.85, 32.44, -64.5) mm, rotated rx 180 ry 0 rz 0.01 deg; joints [27.924, -40.928, 99.012, -148.198, 62.751, 165.202]
  MoveC 7514 to (-327.57, 31.45, -64.5) mm, rotated rx -180 ry 0 rz 0.01 deg; joints [27.914, -40.998, 99.166, -148.231, 62.82, 165.257] to (-325.97, 31.67, -64.5) mm, rotated rx 180 ry 0 rz 0.01 deg; joints [27.949, -41.057, 99.294, -148.212, 62.888, 165.28]
  MoveL 7515 to (-217.36, 95.08, -64.5) mm, rotated rx -180 ry 0 rz 0.01 deg; joints [32.082, -43.792, 105.184, -144.644, 66.664, 165.294]
  MoveC 7516 to (-211.85, 96.65, -64.5) mm, rotated rx 180 ry 0 rz 0.01 deg; joints [32.246, -43.952, 105.535, -144.52, 66.866, 165.345] to (-206.26, 95.45, -64.5) mm, rotated rx 180 ry 0 rz 0.01 deg; joints [32.323, -44.173, 106.027, -144.506, 67.108, 165.484]
  MoveC 7517 to (-201.78, 91.96, -64.5) mm, rotated rx -180 ry 0 rz 0.01 deg; joints [32.301, -44.402, 106.542, -144.599, 67.335, 165.673] to (-199.08, 86.97, -64.5) mm, rotated rx -180 ry 0 rz 0.01 deg; joints [32.193, -44.599, 106.991, -144.772, 67.511, 165.875]
  MoveC 7518 to (-198.79, 85.66, -64.5) mm, rotated rx 180 ry 0 rz 0.01 deg; joints [32.155, -44.637, 107.077, -144.823, 67.54, 165.92] to (-198.7, 84.31, -64.5) mm, rotated rx 180 ry 0 rz 0.01 deg; joints [32.113, -44.668, 107.149, -144.877, 67.563, 165.963]
  MoveL 7519 to (-199.06, 38.43, -64.5) mm, rotated rx -180 ry 0 rz 0.01 deg; joints [30.557, -45.571, 109.261, -146.778, 68.167, 167.325]
  MoveC 7520 to (-200.01, 33.67, -64.5) mm, rotated rx -180 ry 0 rz 0.01 deg; joints [30.374, -45.63, 109.403, -146.987, 68.192, 167.447] to (-201.87, 29.18, -64.5) mm, rotated rx 180 ry 0 rz 0.01 deg; joints [30.182, -45.652, 109.46, -147.195, 68.177, 167.545]
  MoveC 7521 to (-204.65, 25.19, -64.5) mm, rotated rx -180 ry 0 rz 0.01 deg; joints [29.989, -45.631, 109.423, -147.394, 68.116, 167.612] to (-208.29, 21.96, -64.5) mm, rotated rx 180 ry 0 rz 0.01 deg; joints [29.805, -45.567, 109.285, -147.571, 68.011, 167.644]
  MoveC 7522 to (-209.02, 21.51, -64.5) mm, rotated rx -180 ry 0 rz 0.01 deg; joints [29.775, -45.55, 109.249, -147.598, 67.987, 167.644] to (-209.78, 21.12, -64.5) mm, rotated rx -180 ry 0 rz 0.01 deg; joints [29.747, -45.531, 109.208, -147.623, 67.961, 167.643]
  MoveL 7523 to (-309.43, -23.25, -64.5) mm, rotated rx 180 ry 0 rz 0.01 deg; joints [26.399, -42.73, 103.074, -150.418, 64.296, 167.241]
  MoveC 7524 to (-310.21, -24.81, -64.5) mm, rotated rx -180 ry 0 rz 0.01 deg; joints [26.332, -42.728, 103.072, -150.489, 64.28, 167.273] to (-308.85, -25.91, -64.5) mm, rotated rx -180 ry 0 rz 0.01 deg; joints [26.318, -42.8, 103.232, -150.526, 64.354, 167.328]
  MoveL 7525 to (-84.67, -25.91, -64.5) mm, rotated rx -180 ry 0 rz 0.01 deg; joints [30.678, -50.411, 120.501, -147.852, 73.581, 170.94]
  MoveC 7526 to (-83.31, -24.81, -64.5) mm, rotated rx -180 ry 0 rz 0.01 deg; joints [30.75, -50.433, 120.551, -147.783, 73.618, 170.933] to (-84.1, -23.25, -64.5) mm, rotated rx 180 ry 0 rz 0.01 deg; joints [30.791, -50.383, 120.429, -147.73, 73.565, 170.881]
  MoveL 7527 to (-183.96, 21.25, -64.5) mm, rotated rx 180 ry 0 rz 0.01 deg; joints [30.269, -46.409, 111.182, -147.309, 69.008, 168.071]
  MoveC 7528 to (-188.14, 24.08, -64.5) mm, rotated rx 180 ry 0 rz 0.01 deg; joints [30.283, -46.215, 110.739, -147.243, 68.802, 167.921] to (-191.13, 28.15, -64.5) mm, rotated rx -180 ry 0 rz 0.01 deg; joints [30.363, -46.038, 110.33, -147.11, 68.626, 167.755]
  MoveC 7529 to (-193.05, 32.75, -64.5) mm, rotated rx 180 ry 0 rz 0.01 deg; joints [30.484, -45.885, 109.978, -146.942, 68.487, 167.591] to (-194.33, 37.56, -64.5) mm, rotated rx 180 ry 0 rz 0.01 deg; joints [30.623, -45.75, 109.663, -146.757, 68.37, 167.43]
  MoveC 7530 to (-194.67, 39.89, -64.5) mm, rotated rx 180 ry 0 rz 0.01 deg; joints [30.696, -45.693, 109.532, -146.665, 68.325, 167.357] to (-194.78, 42.23, -64.5) mm, rotated rx 180 ry 0 rz 0.01 deg; joints [30.774, -45.644, 109.416, -146.569, 68.289, 167.287]
  MoveL 7531 to (-194.81, 84.32, -64.5) mm, rotated rx 180 ry 0 rz 0.01 deg; joints [32.194, -44.801, 107.446, -144.831, 67.718, 166.032]
  MoveC 7532 to (-193.08, 90.61, -64.5) mm, rotated rx 180 ry 0 rz 0.01 deg; joints [32.439, -44.73, 107.276, -144.552, 67.702, 165.87] to (-188.35, 95.1, -64.5) mm, rotated rx -180 ry 0 rz 0.01 deg; joints [32.688, -44.798, 107.417, -144.311, 67.829, 165.816]
  MoveC 7533 to (-182.04, 96.63, -64.5) mm, rotated rx 180 ry 0 rz 0.01 deg; joints [32.872, -44.981, 107.822, -144.172, 68.058, 165.882] to (-175.78, 94.9, -64.5) mm, rotated rx -180 ry 0 rz 0.01 deg; joints [32.949, -45.229, 108.379, -144.164, 68.33, 166.047]
  MoveL 7534 to (-67.54, 31.67, -64.5) mm, rotated rx 180 ry 0 rz 0.01 deg; joints [33.201, -49.909, 119.186, -145.136, 73.387, 169.71]
  MoveC 7535 to (-65.94, 31.46, -64.5) mm, rotated rx -180 ry 0 rz 0.01 deg; joints [33.231, -49.961, 119.307, -145.117, 73.45, 169.742] to (-64.66, 32.44, -64.5) mm, rotated rx -180 ry 0 rz 0.01 deg; joints [33.298, -49.981, 119.352, -145.054, 73.484, 169.737]
  MoveL 7536 to (-64.22, 33.19, -64.5) mm, rotated rx -180 ry 0 rz 0.01 deg; joints [33.335, -49.98, 119.348, -145.015, 73.489, 169.724]
  MoveC 7537 to (-64.01, 34.8, -64.5) mm, rotated rx 180 ry 0 rz 0.01 deg; joints [33.398, -49.957, 119.289, -144.944, 73.473, 169.684] to (-65, 36.08, -64.5) mm, rotated rx -180 ry 0 rz 0.01 deg; joints [33.421, -49.903, 119.162, -144.908, 73.417, 169.632]
  MoveL 7538 to (-174.23, 98.45, -64.5) mm, rotated rx 180 ry 0 rz 0.01 deg; joints [33.1, -45.207, 108.323, -144, 68.342, 165.965]
  MoveC 7539 to (-178.43, 102.56, -64.5) mm, rotated rx -180 ry 0 rz 0.01 deg; joints [33.146, -44.978, 107.804, -143.884, 68.12, 165.764] to (-180.12, 108.19, -64.5) mm, rotated rx -180 ry 0 rz 0.01 deg; joints [33.295, -44.801, 107.399, -143.675, 67.975, 165.559]
  MoveC 7540 to (-179.12, 113.93, -64.5) mm, rotated rx 180 ry 0 rz 0.01 deg; joints [33.504, -44.712, 107.189, -143.429, 67.936, 165.398] to (-175.86, 118.75, -64.5) mm, rotated rx -180 ry 0 rz 0.01 deg; joints [33.732, -44.719, 107.194, -143.192, 67.998, 165.305]
  MoveC 7541 to (-175, 119.48, -64.5) mm, rotated rx -180 ry 0 rz 0.01 deg; joints [33.775, -44.732, 107.222, -143.152, 68.021, 165.298] to (-174.07, 120.09, -64.5) mm, rotated rx -180 ry 0 rz 0.01 deg; joints [33.815, -44.75, 107.262, -143.115, 68.049, 165.296]
  MoveL 7542 to (-133.77, 142.83, -64.5) mm, rotated rx 180 ry 0 rz 0.01 deg; joints [35.458, -45.586, 109.084, -141.655, 69.286, 165.308]
  MoveC 7543 to (-129.3, 144.29, -64.5) mm, rotated rx 180 ry 0 rz 0.01 deg; joints [35.609, -45.698, 109.333, -141.532, 69.435, 165.342] to (-124.64, 144.84, -64.5) mm, rotated rx -180 ry 0 rz 0.01 deg; joints [35.736, -45.837, 109.642, -141.442, 69.603, 165.409]
  MoveC 7544 to (-119.95, 144.39, -64.5) mm, rotated rx 180 ry 0 rz 0.01 deg; joints [35.83, -45.997, 110.003, -141.391, 69.786, 165.507] to (-115.49, 142.88, -64.5) mm, rotated rx 180 ry 0 rz 0.01 deg; joints [35.886, -46.173, 110.401, -141.385, 69.975, 165.635]
  MoveC 7545 to (-114.74, 142.48, -64.5) mm, rotated rx 180 ry 0 rz 0.01 deg; joints [35.891, -46.206, 110.475, -141.39, 70.008, 165.661] to (-114.03, 142.02, -64.5) mm, rotated rx 180 ry 0 rz 0.01 deg; joints [35.893, -46.238, 110.55, -141.397, 70.042, 165.688]
  MoveL 7546 to (-1.2, 60.25, -64.5) mm, rotated rx 180 ry 0 rz 0.01 deg; joints [35.889, -51.287, 122.362, -142.698, 75.376, 170.044]
  MoveC 7547 to (-0.37, 59.55, -64.5) mm, rotated rx 180 ry 0 rz 0.01 deg; joints [35.885, -51.324, 122.451, -142.71, 75.417, 170.078] to (0.4, 58.77, -64.5) mm, rotated rx 180 ry 0 rz 0.01 deg; joints [35.877, -51.36, 122.538, -142.726, 75.456, 170.112]
  MoveC 7548 to (1.14, 57.98, -64.5) mm, rotated rx -180 ry 0 rz 0.01 deg; joints [35.868, -51.396, 122.625, -142.743, 75.495, 170.146] to (1.93, 57.22, -64.5) mm, rotated rx -180 ry 0 rz 0.01 deg; joints [35.861, -51.432, 122.713, -142.758, 75.535, 170.181]
  MoveC 7549 to (3.85, 56.9, -64.5) mm, rotated rx -180 ry 0 rz 0.01 deg; joints [35.9, -51.491, 122.855, -142.732, 75.609, 170.222] to (4.92, 58.53, -64.5) mm, rotated rx 180 ry 0 rz 0.01 deg; joints [35.987, -51.49, 122.848, -142.643, 75.621, 170.196]
  MoveL 7550 to (4.91, 330, -64.5) mm, rotated rx 180 ry 0 rz 0.01 deg; joints [44.67, -45.163, 107.813, -132.149, 71.517, 161.464]
  MoveC 7551 to (3.78, 332.72, -64.5) mm, rotated rx -180 ry 0 rz 0.01 deg; joints [44.715, -45.055, 107.568, -132.07, 71.44, 161.342] to (1.06, 333.85, -64.5) mm, rotated rx 180 ry 0 rz 0.01 deg; joints [44.671, -44.945, 107.321, -132.079, 71.334, 161.249]
  MoveL 7552 to (-155.01, 333.85, -64.5) mm, rotated rx -180 ry 0 rz 0.01 deg; joints [40.677, -39.99, 96.455, -134.379, 65.805, 158.122]
  MoveC 7553 to (-156.63, 332.74, -64.5) mm, rotated rx 180 ry 0 rz 0.01 deg; joints [40.608, -39.966, 96.404, -134.44, 65.759, 158.13] to (-156.2, 330.82, -64.5) mm, rotated rx 180 ry 0 rz 0.01 deg; joints [40.565, -40.037, 96.561, -134.51, 65.802, 158.215]
  MoveC 7554 to (-154.61, 329.36, -64.5) mm, rotated rx 180 ry 0 rz 0.01 deg; joints [40.562, -40.135, 96.775, -134.55, 65.883, 158.307] to (-152.99, 327.92, -64.5) mm, rotated rx -180 ry 0 rz 0.01 deg; joints [40.561, -40.232, 96.988, -134.588, 65.964, 158.399]
  MoveC 7555 to (-151.48, 326.36, -64.5) mm, rotated rx 180 ry 0 rz 0.01 deg; joints [40.553, -40.329, 97.202, -134.633, 66.042, 158.492] to (-150.25, 324.58, -64.5) mm, rotated rx -180 ry 0 rz 0.01 deg; joints [40.533, -40.423, 97.408, -134.689, 66.113, 158.588]
  MoveC 7556 to (-147.39, 319.49, -64.5) mm, rotated rx 180 ry 0 rz 0.01 deg; joints [40.459, -40.667, 97.945, -134.855, 66.291, 158.847] to (-144.61, 314.36, -64.5) mm, rotated rx -180 ry 0 rz 0.01 deg; joints [40.382, -40.908, 98.476, -135.023, 66.467, 159.103]
  MoveC 7557 to (-142.32, 308.97, -64.5) mm, rotated rx -180 ry 0 rz 0.01 deg; joints [40.285, -41.138, 98.985, -135.206, 66.628, 159.357] to (-141, 303.27, -64.5) mm, rotated rx 180 ry 0 rz 0.01 deg; joints [40.155, -41.342, 99.439, -135.413, 66.757, 159.602]
  MoveL 7558 to (-126.98, 164.32, -64.5) mm, rotated rx -180 ry 0 rz 0.01 deg; joints [36.307, -45.321, 108.451, -140.697, 69.238, 164.743]
  MoveC 7559 to (-127.43, 158.88, -64.5) mm, rotated rx -180 ry 0 rz 0.01 deg; joints [36.122, -45.431, 108.706, -140.921, 69.298, 164.911] to (-129.8, 153.95, -64.5) mm, rotated rx -180 ry 0 rz 0.01 deg; joints [35.909, -45.465, 108.793, -141.152, 69.279, 165.025]
  MoveC 7560 to (-133.25, 149.82, -64.5) mm, rotated rx 180 ry 0 rz 0.01 deg; joints [35.696, -45.447, 108.759, -141.367, 69.207, 165.095] to (-137.2, 146.16, -64.5) mm, rotated rx 180 ry 0 rz 0.01 deg; joints [35.487, -45.4, 108.662, -141.57, 69.109, 165.14]
  MoveC 7561 to (-137.84, 145.66, -64.5) mm, rotated rx 180 ry 0 rz 0.01 deg; joints [35.456, -45.39, 108.641, -141.599, 69.091, 165.144] to (-138.5, 145.19, -64.5) mm, rotated rx -180 ry 0 rz 0.01 deg; joints [35.426, -45.379, 108.617, -141.627, 69.073, 165.147]
  MoveC 7562 to (-139.17, 144.74, -64.5) mm, rotated rx 180 ry 0 rz 0.01 deg; joints [35.396, -45.367, 108.591, -141.654, 69.053, 165.149] to (-139.87, 144.33, -64.5) mm, rotated rx 180 ry 0 rz 0.01 deg; joints [35.367, -45.354, 108.562, -141.681, 69.033, 165.15]
  MoveL 7563 to (-176.15, 123.35, -64.5) mm, rotated rx 180 ry 0 rz 0.01 deg; joints [33.876, -44.609, 106.941, -143.009, 67.923, 165.155]
  MoveC 7564 to (-181.6, 121.77, -64.5) mm, rotated rx 180 ry 0 rz 0.01 deg; joints [33.706, -44.458, 106.609, -143.14, 67.73, 165.106] to (-187.16, 122.91, -64.5) mm, rotated rx -180 ry 0 rz 0.01 deg; joints [33.623, -44.243, 106.129, -143.161, 67.495, 164.968]
  MoveC 7565 to (-191.63, 126.33, -64.5) mm, rotated rx -180 ry 0 rz 0.01 deg; joints [33.637, -44.014, 105.615, -143.075, 67.271, 164.777] to (-194.38, 131.24, -64.5) mm, rotated rx 180 ry 0 rz 0.01 deg; joints [33.736, -43.811, 105.155, -142.907, 67.095, 164.568]
  MoveC 7566 to (-194.69, 132.61, -64.5) mm, rotated rx -180 ry 0 rz 0.01 deg; joints [33.773, -43.769, 105.061, -142.855, 67.064, 164.518] to (-194.8, 134.02, -64.5) mm, rotated rx -180 ry 0 rz 0.01 deg; joints [33.816, -43.734, 104.981, -142.799, 67.04, 164.471]
  MoveL 7567 to (-194.21, 259.89, -64.5) mm, rotated rx -180 ry 0 rz 0.01 deg; joints [37.675, -40.676, 98.058, -137.719, 65.328, 160.116]
  MoveC 7568 to (-194.82, 261.38, -64.5) mm, rotated rx 180 ry 0 rz 0.01 deg; joints [37.704, -40.614, 97.921, -137.666, 65.283, 160.048] to (-196.32, 262, -64.5) mm, rotated rx -180 ry 0 rz 0.01 deg; joints [37.689, -40.544, 97.768, -137.656, 65.216, 159.993]
  MoveL 7569 to (-197.19, 262, -64.5) mm, rotated rx 180 ry 0 rz 0.01 deg; joints [37.669, -40.513, 97.7, -137.665, 65.182, 159.974]
  MoveC 7570 to (-198.69, 261.38, -64.5) mm, rotated rx 180 ry 0 rz 0.01 deg; joints [37.618, -40.476, 97.621, -137.704, 65.132, 159.966] to (-199.31, 259.89, -64.5) mm, rotated rx 180 ry 0 rz 0.01 deg; joints [37.56, -40.494, 97.662, -137.77, 65.128, 160.008]
  MoveL 7571 to (-198.71, 134.02, -64.5) mm, rotated rx -180 ry 0 rz 0.01 deg; joints [33.732, -43.598, 104.681, -142.844, 66.885, 164.398]
  MoveC 7572 to (-200.1, 128.5, -64.5) mm, rotated rx 180 ry 0 rz 0.01 deg; joints [33.526, -43.673, 104.855, -143.084, 66.905, 164.55] to (-203.93, 124.3, -64.5) mm, rotated rx 180 ry 0 rz 0.01 deg; joints [33.31, -43.632, 104.773, -143.299, 66.809, 164.614]
  MoveC 7573 to (-209.16, 122.21, -64.5) mm, rotated rx 180 ry 0 rz 0.01 deg; joints [33.132, -43.495, 104.475, -143.442, 66.628, 164.584] to (-214.79, 122.33, -64.5) mm, rotated rx 180 ry 0 rz 0.01 deg; joints [33.018, -43.294, 104.031, -143.498, 66.4, 164.475]
  MoveC 7574 to (-215.49, 122.53, -64.5) mm, rotated rx 180 ry 0 rz 0.01 deg; joints [33.01, -43.265, 103.966, -143.498, 66.369, 164.455] to (-216.18, 122.78, -64.5) mm, rotated rx 180 ry 0 rz 0.01 deg; joints [33.004, -43.235, 103.9, -143.495, 66.338, 164.434]
  MoveC 7575 to (-216.85, 123.08, -64.5) mm, rotated rx -180 ry 0 rz 0.01 deg; joints [32.999, -43.205, 103.832, -143.49, 66.307, 164.412] to (-217.5, 123.42, -64.5) mm, rotated rx 180 ry 0 rz 0.01 deg; joints [32.997, -43.174, 103.764, -143.483, 66.276, 164.389]
  MoveL 7576 to (-256.62, 146.38, -64.5) mm, rotated rx -180 ry 0 rz 0.01 deg; joints [32.921, -41.235, 99.47, -142.914, 64.367, 162.87]
  MoveC 7577 to (-260.4, 149.65, -64.5) mm, rotated rx 180 ry 0 rz 0.01 deg; joints [32.946, -41.019, 98.992, -142.811, 64.166, 162.683] to (-263.45, 153.61, -64.5) mm, rotated rx -180 ry 0 rz 0.01 deg; joints [33.008, -40.812, 98.534, -142.673, 63.986, 162.485]
  MoveC 7578 to (-265.56, 158.14, -64.5) mm, rotated rx -180 ry 0 rz 0.01 deg; joints [33.105, -40.625, 98.12, -142.502, 63.837, 162.285] to (-266.54, 163.05, -64.5) mm, rotated rx 180 ry 0 rz 0.01 deg; joints [33.236, -40.472, 97.777, -142.307, 63.731, 162.094]
  MoveC 7579 to (-266.57, 163.87, -64.5) mm, rotated rx 180 ry 0 rz 0.01 deg; joints [33.261, -40.451, 97.731, -142.274, 63.719, 162.065] to (-266.52, 164.69, -64.5) mm, rotated rx 180 ry 0 rz 0.01 deg; joints [33.287, -40.433, 97.691, -142.24, 63.71, 162.037]
  MoveL 7580 to (-252.39, 303.98, -64.5) mm, rotated rx 180 ry 0 rz 0.01 deg; joints [37.652, -37.283, 90.668, -136.406, 62.392, 157.094]
  MoveC 7581 to (-250.76, 309.94, -64.5) mm, rotated rx 180 ry 0 rz 0.01 deg; joints [37.852, -37.172, 90.42, -136.151, 62.376, 156.89] to (-248.56, 315.72, -64.5) mm, rotated rx 180 ry 0 rz 0.01 deg; joints [38.059, -37.086, 90.229, -135.9, 62.386, 156.707]
  MoveC 7582 to (-245.68, 321.2, -64.5) mm, rotated rx 180 ry 0 rz 0.01 deg; joints [38.272, -37.035, 90.111, -135.658, 62.428, 156.551] to (-242.05, 326.21, -64.5) mm, rotated rx 180 ry 0 rz 0.01 deg; joints [38.488, -37.025, 90.083, -135.43, 62.505, 156.431]
  MoveC 7583 to (-240.95, 327.44, -64.5) mm, rotated rx 180 ry 0 rz 0.01 deg; joints [38.546, -37.031, 90.094, -135.372, 62.533, 156.407] to (-239.76, 328.59, -64.5) mm, rotated rx 180 ry 0 rz 0.01 deg; joints [38.603, -37.043, 90.116, -135.318, 62.565, 156.389]
  MoveC 7584 to (-238.54, 329.7, -64.5) mm, rotated rx -180 ry 0 rz 0.01 deg; joints [38.661, -37.056, 90.144, -135.265, 62.6, 156.372] to (-237.32, 330.82, -64.5) mm, rotated rx 180 ry 0 rz 0.01 deg; joints [38.718, -37.069, 90.171, -135.211, 62.633, 156.356]
  MoveC 7585 to (-236.88, 332.74, -64.5) mm, rotated rx -180 ry 0 rz 0.01 deg; joints [38.78, -37.029, 90.08, -135.13, 62.624, 156.286] to (-238.51, 333.85, -64.5) mm, rotated rx -180 ry 0 rz 0.01 deg; joints [38.774, -36.932, 89.873, -135.095, 62.543, 156.201]
  MoveL 7586 to (-394.58, 333.84, -64.5) mm, rotated rx 180 ry 0 rz 0.01 deg; joints [35.598, -30.194, 75.592, -135.203, 55.729, 151.725]
  MoveC 7587 to (-397.3, 332.71, -64.5) mm, rotated rx -180 ry 0 rz 0.01 deg; joints [35.516, -30.099, 75.396, -135.239, 55.616, 151.687] to (-398.43, 329.99, -64.5) mm, rotated rx -180 ry 0 rz 0.01 deg; joints [35.423, -30.137, 75.479, -135.359, 55.602, 151.782]
  MoveL 7588 to (-398.43, 178.86, -64.5) mm, rotated rx 180 ry 0 rz 0.01 deg; joints [31.223, -34.664, 85.273, -142.161, 57.709, 158.468]
  MoveL 7589 to (-398.27, 178.25, -64.33) mm, rotated rx 180 ry 0 rz 0.01 deg; joints [31.208, -34.695, 85.324, -142.185, 57.719, 158.491]
  MoveL 7590 to (-397.98, 177.89, -63.87) mm, rotated rx -180 ry 0 rz 0.01 deg; joints [31.203, -34.739, 85.375, -142.194, 57.723, 158.5]
  MoveL 7591 to (-397.84, 177.79, -63.23) mm, rotated rx 180 ry 0 rz 0.01 deg; joints [31.202, -34.778, 85.399, -142.19, 57.711, 158.49]
  Set speed (1000.0 mm/s)
  MoveL 7592 to (-397.84, 177.79, 11) mm, rotated rx 180 ry 0 rz 0.01 deg; joints [31.164, -38.121, 85.702, -140.981, 55.312, 156.248]
  Set speed (1000.0 mm/s)
  MoveL 7593 to (-397.45, 339.19, 11) mm, rotated rx -180 ry 0 rz 0.01 deg; joints [35.652, -33.08, 75.236, -133.498, 53.489, 148.847]
  Set speed (100.0 mm/s)
  MoveL 7594 to (-397.45, 339.19, -42.73) mm, rotated rx -180 ry 0 rz 0.01 deg; joints [35.675, -30.82, 75.053, -134.55, 54.945, 150.674]
  MoveL 7595 to (-397.51, 339.2, -43.12) mm, rotated rx 180 ry 0 rz 0.01 deg; joints [35.674, -30.8, 75.044, -134.557, 54.953, 150.684]
  MoveL 7596 to (-397.69, 339.2, -43.48) mm, rotated rx 180 ry 0 rz 0.01 deg; joints [35.671, -30.775, 75.023, -134.562, 54.953, 150.689]
  MoveL 7597 to (-398.51, 339.2, -43.98) mm, rotated rx -180 ry 0 rz 0.01 deg; joints [35.656, -30.713, 74.936, -134.566, 54.928, 150.677]
  MoveL 7598 to (-398.67, 339.2, -44) mm, rotated rx -180 ry 0 rz 0.01 deg; joints [35.652, -30.704, 74.919, -134.565, 54.921, 150.672]
  MoveL 7599 to (-399.34, 339.13, -44.02) mm, rotated rx -180 ry 0 rz 0.01 deg; joints [35.638, -30.672, 74.855, -134.564, 54.891, 150.652]
  MoveL 7600 to (-399.55, 339.1, -44.03) mm, rotated rx -180 ry 0 rz 0.01 deg; joints [35.633, -30.663, 74.835, -134.564, 54.881, 150.647]
  MoveL 7601 to (-402.87, 337.02, -44.17) mm, rotated rx 180 ry 0 rz 0.01 deg; joints [35.516, -30.564, 74.645, -134.641, 54.757, 150.639]
  MoveL 7602 to (-402.89, 336.99, -44.17) mm, rotated rx -180 ry 0 rz 0.01 deg; joints [35.515, -30.564, 74.645, -134.642, 54.757, 150.64]
  MoveL 7603 to (-403.36, 336.14, -44.21) mm, rotated rx -180 ry 0 rz 0.01 deg; joints [35.484, -30.569, 74.659, -134.679, 54.747, 150.667]
  MoveL 7604 to (-403.42, 336, -44.21) mm, rotated rx -180 ry 0 rz 0.01 deg; joints [35.479, -30.57, 74.663, -134.686, 54.746, 150.672]
  MoveL 7605 to (-403.6, 335.45, -44.23) mm, rotated rx -180 ry 0 rz 0.01 deg; joints [35.461, -30.58, 74.685, -134.711, 54.746, 150.694]
  MoveL 7606 to (-403.64, 335.28, -44.24) mm, rotated rx 180 ry 0 rz 0.01 deg; joints [35.456, -30.583, 74.693, -134.719, 54.747, 150.701]
  MoveL 7607 to (-403.75, 334.45, -44.27) mm, rotated rx 180 ry 0 rz 0.01 deg; joints [35.432, -30.605, 74.742, -134.758, 54.754, 150.74]
  MoveL 7608 to (-403.78, 333.95, -44.29) mm, rotated rx -180 ry 0 rz 0.01 deg; joints [35.418, -30.621, 74.776, -134.782, 54.76, 150.765]
  MoveL 7609 to (-403.79, 333.65, -44.3) mm, rotated rx -180 ry 0 rz 0.01 deg; joints [35.41, -30.63, 74.797, -134.796, 54.764, 150.78]
  MoveL 7610 to (-403.79, 333.1, -44.31) mm, rotated rx 180 ry 0 rz 0.01 deg; joints [35.396, -30.648, 74.838, -134.822, 54.772, 150.808]
  MoveL 7611 to (-401.27, 328.17, -44.52) mm, rotated rx -180 ry 0 rz 0.01 deg; joints [35.313, -30.934, 75.456, -135.075, 54.965, 151.147]
  MoveL 7612 to (-395.8, 327.3, -44.72) mm, rotated rx -180 ry 0 rz 0.01 deg; joints [35.393, -31.224, 76.077, -135.154, 55.24, 151.383]
  MoveL 7613 to (-391.89, 331.22, -44.92) mm, rotated rx 180 ry 0 rz 0.01 deg; joints [35.571, -31.273, 76.191, -134.999, 55.375, 151.33]
  MoveL 7614 to (-392.75, 336.69, -45.12) mm, rotated rx -180 ry 0 rz 0.01 deg; joints [35.699, -31.034, 75.703, -134.742, 55.264, 151.037]
  MoveL 7615 to (-397.69, 339.2, -45.32) mm, rotated rx -180 ry 0 rz 0.01 deg; joints [35.672, -30.696, 75.012, -134.595, 55.002, 150.748]
  MoveL 7616 to (-398.51, 339.2, -45.35) mm, rotated rx -180 ry 0 rz 0.01 deg; joints [35.656, -30.654, 74.928, -134.59, 54.964, 150.721]
  MoveL 7617 to (-399.34, 339.13, -45.38) mm, rotated rx 180 ry 0 rz 0.01 deg; joints [35.639, -30.614, 74.847, -134.588, 54.927, 150.696]
  MoveL 7618 to (-399.55, 339.1, -45.38) mm, rotated rx -180 ry 0 rz 0.01 deg; joints [35.634, -30.604, 74.827, -134.588, 54.917, 150.69]
  MoveL 7619 to (-402.87, 337.02, -45.52) mm, rotated rx -180 ry 0 rz 0.01 deg; joints [35.517, -30.506, 74.637, -134.666, 54.793, 150.683]
  MoveL 7620 to (-402.89, 336.99, -45.53) mm, rotated rx 180 ry 0 rz 0.01 deg; joints [35.516, -30.506, 74.637, -134.667, 54.792, 150.683]
  MoveL 7621 to (-403.36, 336.14, -45.56) mm, rotated rx -180 ry 0 rz 0.01 deg; joints [35.485, -30.51, 74.651, -134.704, 54.783, 150.71]
  MoveL 7622 to (-403.42, 336, -45.56) mm, rotated rx 180 ry 0 rz 0.01 deg; joints [35.48, -30.512, 74.655, -134.71, 54.782, 150.715]
  MoveL 7623 to (-403.6, 335.45, -45.58) mm, rotated rx -180 ry 0 rz 0.01 deg; joints [35.462, -30.521, 74.676, -134.735, 54.782, 150.737]
  MoveL 7624 to (-403.64, 335.28, -45.59) mm, rotated rx -180 ry 0 rz 0.01 deg; joints [35.457, -30.525, 74.685, -134.743, 54.783, 150.745]
  MoveL 7625 to (-403.75, 334.45, -45.62) mm, rotated rx -180 ry 0 rz 0.01 deg; joints [35.433, -30.547, 74.734, -134.782, 54.789, 150.783]
  MoveL 7626 to (-403.78, 333.95, -45.64) mm, rotated rx -180 ry 0 rz 0.01 deg; joints [35.419, -30.562, 74.768, -134.806, 54.796, 150.808]
  MoveL 7627 to (-403.79, 333.65, -45.65) mm, rotated rx 180 ry 0 rz 0.01 deg; joints [35.411, -30.572, 74.789, -134.82, 54.8, 150.823]
  MoveL 7628 to (-403.79, 333.1, -45.67) mm, rotated rx -180 ry 0 rz 0.01 deg; joints [35.396, -30.59, 74.83, -134.847, 54.808, 150.851]
  MoveL 7629 to (-401.27, 328.17, -45.87) mm, rotated rx -180 ry 0 rz 0.01 deg; joints [35.313, -30.876, 75.448, -135.1, 55.001, 151.19]
  MoveL 7630 to (-395.8, 327.3, -46.07) mm, rotated rx 180 ry 0 rz 0.01 deg; joints [35.393, -31.165, 76.069, -135.178, 55.276, 151.426]
  MoveL 7631 to (-391.89, 331.22, -46.27) mm, rotated rx -180 ry 0 rz 0.01 deg; joints [35.571, -31.214, 76.183, -135.023, 55.411, 151.373]
  MoveL 7632 to (-392.75, 336.69, -46.47) mm, rotated rx 180 ry 0 rz 0.01 deg; joints [35.699, -30.976, 75.695, -134.766, 55.299, 151.081]
  MoveL 7633 to (-397.69, 339.2, -46.67) mm, rotated rx 180 ry 0 rz 0.01 deg; joints [35.672, -30.637, 75.004, -134.62, 55.038, 150.792]
  MoveL 7634 to (-398.51, 339.2, -46.7) mm, rotated rx 180 ry 0 rz 0.01 deg; joints [35.657, -30.595, 74.919, -134.615, 55, 150.764]
  MoveL 7635 to (-399.34, 339.13, -46.73) mm, rotated rx -180 ry 0 rz 0.01 deg; joints [35.639, -30.555, 74.839, -134.613, 54.962, 150.739]
  MoveL 7636 to (-399.55, 339.1, -46.74) mm, rotated rx -180 ry 0 rz 0.01 deg; joints [35.634, -30.546, 74.819, -134.613, 54.953, 150.734]
  MoveL 7637 to (-402.87, 337.02, -46.88) mm, rotated rx -180 ry 0 rz 0.01 deg; joints [35.517, -30.447, 74.629, -134.69, 54.829, 150.726]
  MoveL 7638 to (-402.89, 336.99, -46.88) mm, rotated rx -180 ry 0 rz 0.01 deg; joints [35.516, -30.447, 74.629, -134.691, 54.828, 150.727]
  MoveL 7639 to (-403.36, 336.14, -46.91) mm, rotated rx -180 ry 0 rz 0.01 deg; joints [35.485, -30.452, 74.642, -134.729, 54.819, 150.754]
  MoveL 7640 to (-403.42, 336, -46.92) mm, rotated rx -180 ry 0 rz 0.01 deg; joints [35.48, -30.453, 74.646, -134.735, 54.818, 150.759]
  MoveL 7641 to (-403.6, 335.45, -46.94) mm, rotated rx 180 ry 0 rz 0.01 deg; joints [35.463, -30.463, 74.668, -134.76, 54.817, 150.781]
  MoveL 7642 to (-403.64, 335.28, -46.94) mm, rotated rx -180 ry 0 rz 0.01 deg; joints [35.457, -30.466, 74.677, -134.768, 54.818, 150.788]
  MoveL 7643 to (-403.75, 334.45, -46.97) mm, rotated rx 180 ry 0 rz 0.01 deg; joints [35.433, -30.488, 74.726, -134.807, 54.825, 150.827]
  MoveL 7644 to (-403.78, 333.95, -46.99) mm, rotated rx -180 ry 0 rz 0.01 deg; joints [35.419, -30.504, 74.76, -134.831, 54.831, 150.851]
  MoveL 7645 to (-403.79, 333.65, -47) mm, rotated rx -180 ry 0 rz 0.01 deg; joints [35.412, -30.513, 74.781, -134.845, 54.835, 150.866]
  MoveL 7646 to (-403.79, 333.1, -47.02) mm, rotated rx 180 ry 0 rz 0.01 deg; joints [35.397, -30.531, 74.821, -134.871, 54.844, 150.894]
  MoveL 7647 to (-401.27, 328.17, -47.22) mm, rotated rx 180 ry 0 rz 0.01 deg; joints [35.314, -30.817, 75.44, -135.124, 55.037, 151.233]
  MoveL 7648 to (-395.8, 327.3, -47.42) mm, rotated rx 180 ry 0 rz 0.01 deg; joints [35.394, -31.106, 76.061, -135.203, 55.312, 151.469]
  MoveL 7649 to (-391.89, 331.22, -47.62) mm, rotated rx 180 ry 0 rz 0.01 deg; joints [35.572, -31.155, 76.174, -135.047, 55.447, 151.416]
  MoveL 7650 to (-392.75, 336.69, -47.82) mm, rotated rx -180 ry 0 rz 0.01 deg; joints [35.7, -30.917, 75.687, -134.79, 55.335, 151.124]
  MoveL 7651 to (-397.69, 339.2, -48.02) mm, rotated rx 180 ry 0 rz 0.01 deg; joints [35.673, -30.578, 74.995, -134.644, 55.073, 150.835]
  MoveL 7652 to (-398.51, 339.2, -48.05) mm, rotated rx 180 ry 0 rz 0.01 deg; joints [35.657, -30.537, 74.911, -134.639, 55.035, 150.807]
  MoveL 7653 to (-399.34, 339.13, -48.08) mm, rotated rx -180 ry 0 rz 0.01 deg; joints [35.64, -30.497, 74.83, -134.637, 54.998, 150.783]
  MoveL 7654 to (-399.55, 339.1, -48.09) mm, rotated rx 180 ry 0 rz 0.01 deg; joints [35.635, -30.487, 74.81, -134.637, 54.988, 150.777]
  MoveL 7655 to (-402.87, 337.02, -48.23) mm, rotated rx 180 ry 0 rz 0.01 deg; joints [35.518, -30.389, 74.62, -134.715, 54.864, 150.769]
  MoveL 7656 to (-402.89, 336.99, -48.23) mm, rotated rx -180 ry 0 rz 0.01 deg; joints [35.517, -30.389, 74.62, -134.716, 54.864, 150.77]
  MoveL 7657 to (-403.36, 336.14, -48.26) mm, rotated rx 180 ry 0 rz 0.01 deg; joints [35.486, -30.393, 74.634, -134.753, 54.854, 150.797]
  MoveL 7658 to (-403.42, 336, -48.27) mm, rotated rx 180 ry 0 rz 0.01 deg; joints [35.481, -30.395, 74.638, -134.759, 54.853, 150.802]
  MoveL 7659 to (-403.6, 335.45, -48.29) mm, rotated rx -180 ry 0 rz 0.01 deg; joints [35.463, -30.404, 74.66, -134.784, 54.853, 150.824]
